    _RailLengthXpu                := _fbXpuPart.GetLength();
    _RailLengthGroup              := _fbMc2CaGroup.GetRailLength();
    _nLengthXpu                   := TO_UINT(_RailLengthXpu);
    _nLengthGroup                 := TO_UINT(_RailLengthGroup);
END_CASE
//-----------------------------------------------------------------------------
//-----------------------------------------------------------------------------
CASE _eState
OF
  //---------------------------------------------------------------------------
  E_PROGRESS.PROGRESS_STARTUP:    // check data for errors
    IF NOT (_bAllPositionsValid)
    THEN
      _eChk                       := E_XPU_CHECK.PROCESSING_UNIT_POSITIONS_VALID;
      _eState := _eResult         := E_PROGRESS.PROGRESS_ERROR;

      _stMsg.eType                := E_MessageType.eMessageError;
      _stMsg.eSubdevice           := e_Subdevice.Xpu_fbProcessingUnit;
      _stMsg.iErrorNumber         := 0;
      _stMsg.sText                := concat(TO_STRING(E_XPU_CHECK.PROCESSING_UNIT_POSITIONS_VALID), ': ');
      _stMsg.sText                := concat(_stMsg.sText, TO_STRING(_eResult));
      f_MessageSet(_stMsg);

    ELSIF NOT (_nLengthXpu > 0)
    THEN
      _eChk                       := E_XPU_CHECK.XPU_RAIL_LENGTH;
      _eState := _eResult         := E_PROGRESS.PROGRESS_ERROR;

      _stMsg.eType                := E_MessageType.eMessageError;
      _stMsg.eSubdevice           := e_Subdevice.Xpu_fbProcessingUnit;
      _stMsg.iErrorNumber         := 0;
      _stMsg.sText                := concat(TO_STRING(E_XPU_CHECK.XPU_RAIL_LENGTH), ': ');
      _stMsg.sText                := concat(_stMsg.sText, TO_STRING(_eResult));
      f_MessageSet(_stMsg);

    ELSIF NOT (_nLengthGroup > 0)
    THEN
      _eChk                       := E_XPU_CHECK.GROUP_RAIL_LENGTH;
      _eState := _eResult         := E_PROGRESS.PROGRESS_ERROR;
     
      _stMsg.eType                := E_MessageType.eMessageError;
      _stMsg.eSubdevice           := e_Subdevice.Xpu_fbProcessingUnit;
      _stMsg.iErrorNumber         := 0;
      _stMsg.sText                := concat(TO_STRING(E_XPU_CHECK.GROUP_RAIL_LENGTH), ': ');
      _stMsg.sText                := concat(_stMsg.sText, TO_STRING(_eResult));
      f_MessageSet(_stMsg);

    ELSIF NOT (_nDetectedMoverCount = _nExpectedMoverCount)
    THEN
      _bMoverIdDetectionValid     := FALSE;
      _eChk                       := E_XPU_CHECK.MOVER_COUNT_NOT_EQUAL;
      _eState := _eResult         := E_PROGRESS.PROGRESS_ERROR;

      _stMsg.eType                := E_MessageType.eMessageError;
      _stMsg.eSubdevice           := e_Subdevice.Xpu_fbProcessingUnit;
      _stMsg.iErrorNumber         := 0;
      _stMsg.sText                := concat(TO_STRING(E_XPU_CHECK.MOVER_COUNT_NOT_EQUAL), ': ');
      _stMsg.sText                := concat(_stMsg.sText, TO_STRING(_eResult));
      f_MessageSet(_stMsg);
  
    ELSIF NOT (_nLengthXpu = _nLengthGroup)
    THEN
      _eChk                       := E_XPU_CHECK.RAIL_LENGTH_COMPARE;
      _eState := _eResult         := E_PROGRESS.PROGRESS_ERROR;
 
      _stMsg.eType                := E_MessageType.eMessageError;
      _stMsg.eSubdevice           := e_Subdevice.Xpu_fbProcessingUnit;
      _stMsg.iErrorNumber         := 0;
      _stMsg.sText                := concat(TO_STRING(E_XPU_CHECK.RAIL_LENGTH_COMPARE), ': ');
      _stMsg.sText                := concat(_stMsg.sText, TO_STRING(_eResult));
      f_MessageSet(_stMsg);

    ELSE
      _eResult                    := E_PROGRESS.PROGRESS_WORKING;

      IF NOT (__ISVALIDREF(_ModuleInfoData))
      THEN
        _eState                   := E_PROGRESS.PROGRESS_BUSY;

        _stMsg.eType              := E_MessageType.eMessageError;
        _stMsg.eSubdevice         := e_Subdevice.Xpu_fbPartModules;
        _stMsg.iErrorNumber       := 0;
        _stMsg.sText              := concat(TO_STRING(_eState), ': ');
        _stMsg.sText              := concat(_stMsg.sText, 'NOT VALID _ModuleInfoData ref');
      ELSE
        _eJobResult               := ModuleInfoData(TRUE);
  
        IF (_eJobResult = E_PROGRESS.PROGRESS_DONE)
        THEN
          _eState                 := E_PROGRESS.PROGRESS_BUSY;
        END_IF  
      END_IF
    END_IF
END_CASE

Cycle                             := _eResult;
END_METHOD

METHOD GetEnvironment : I_TcIoXtsEnvironment
VAR_INPUT
END_VAR
IF NOT (_eInit = E_XPU_INIT.INIT_DONE) THEN RETURN; END_IF

GetEnvironment := _fbEnvironment;
END_METHOD

METHOD GetNctBaseUnit : Tc3_XTS_Utility.I_TcIoXtsNctBaseUnitInterface
VAR_INPUT
  Index     : UINT;
END_VAR
IF NOT (_eInit = E_XPU_INIT.INIT_DONE) THEN RETURN; END_IF

IF NOT (Index > 0) OR
   NOT (Index < MAX_NCT_BASE_UNIT+1)
THEN
  RETURN;
ELSE
  GetNctBaseUnit    := _ItfNctBaseUnit[Index];
END_IF
END_METHOD

METHOD GetNctController : Tc3_XTS_Utility.I_TcIoXtsNctController
VAR_INPUT
END_VAR
IF NOT (_eInit = E_XPU_INIT.INIT_DONE) THEN RETURN; END_IF

GetNctController := _fbNctController;
END_METHOD

METHOD GetParameterSet : I_TcIoXtsParameterSet
VAR_INPUT
  Index     : UINT;
END_VAR
IF NOT (_eInit = E_XPU_INIT.INIT_DONE) THEN RETURN; END_IF

IF NOT (Index > 0) OR
   NOT (Index < MAX_PARAMETER_SET+1)
THEN
  RETURN;
ELSE
  GetParameterSet   := _fbParameterSet[Index];
END_IF
END_METHOD

METHOD GetProcessingUnit : Tc3_XTS_Utility.I_TcIoXtsProcessingUnit
VAR_INPUT
END_VAR
IF NOT (_eInit = E_XPU_INIT.INIT_DONE) THEN RETURN; END_IF

GetProcessingUnit := _fbProcessingUnit;
END_METHOD

METHOD GetXpuMover : Tc3_XTS_Utility.I_TcIoXtsXpuMover
VAR_INPUT
  Index     : UINT;
END_VAR
IF NOT (_eInit = E_XPU_INIT.INIT_DONE) THEN RETURN; END_IF

IF NOT (Index > 0) OR
   NOT (Index < MAX_MOVER+1)
THEN
  RETURN;
ELSE
  GetXpuMover   := _fbMoverXpu[Index];
END_IF
END_METHOD

// mothers' little helper for display in visu
METHOD IdDetectionModeToString : string(20)
VAR
  _DetectionMode    : MoverIdDetectionMode; // Mover ID detection procedure
END_VAR
// just a little helper for visu display
IF NOT (_eInit = E_XPU_INIT.INIT_DONE) THEN IdDetectionModeToString := 'INIT required'; RETURN; END_IF

_DetectionMode := _fbProcessingUnit.GetMoverIdDetectionMode();

CASE _DetectionMode
OF
  MoverIdDetectionMode.Standard:
    IdDetectionModeToString       := 'Standard';

  MoverIdDetectionMode.Mover1:
    IdDetectionModeToString       := 'Mover 1';

  MoverIdDetectionMode.MultipleMover1:
    IdDetectionModeToString       := 'Multiple Mover 1';

ELSE
    IdDetectionModeToString       := 'UNKNOWN Mode';
END_CASE
END_METHOD

PROPERTY MessageLevel : e_messagetype
SET
_eMessageLevel := MessageLevel;
END_SET
END_PROPERTY

// mothers' little helper for display in visu
METHOD PRIVATE ModuleInfoData : E_PROGRESS
VAR_INPUT
  Enable        : BOOL; // enable to read ST_InfoDataView for diag/display
END_VAR
VAR_INST
  _idt,
  _nModule : UINT;
  _eReturn,
  _eState       : E_PROGRESS;
  _aPcbTemp     : ARRAY[1..4] OF REAL;
END_VAR
//---------------------------------------------------------------------------------------------
// just a little helper for visu display
// collects module data for local data
//---------------------------------------------------------------------------------------------
IF NOT (_eInit = E_XPU_INIT.INIT_DONE)      // if Xpu init is not done, just leave
THEN 
  RETURN; 
END_IF
//---------------------------------------------------------------------------------------------
IF NOT Enable                               // clear states on request
THEN
  _eReturn                                  := 
  _eState                                   := E_PROGRESS.PROGRESS_INIT; 
END_IF 
//---------------------------------------------------------------------------------------------
IF NOT (__ISVALIDREF(_ModuleInfoData))      // datafield not connected, error and leave
THEN
  ModuleInfoData                            := E_PROGRESS.PROGRESS_ERROR;
  RETURN;
END_IF
//---------------------------------------------------------------------------------------------
CASE _eState                                // get InfoData from motor modules
OF
  //-------------------------------------------------------------------------------------------
  E_PROGRESS.PROGRESS_INIT:
    IF Enable
    THEN
      _eState                                             := E_PROGRESS.PROGRESS_BUSY;
      _nModule                                            := 1;
    END_IF
END_CASE
CASE _eState
OF
  //-------------------------------------------------------------------------------------------
  E_PROGRESS.PROGRESS_BUSY:
    _eState                                               := E_PROGRESS.PROGRESS_PREPARE;

    _ModuleInfoData[_nModule].fAuxiliaryVoltage_5V        := _fbPartModules[_nModule].GetAuxiliaryVoltage5V();
    _ModuleInfoData[_nModule].fAuxiliaryVoltage_10V       := _fbPartModules[_nModule].GetAuxiliaryVoltage10V();
    _ModuleInfoData[_nModule].fAuxiliaryVoltage_24V       := _fbPartModules[_nModule].GetAuxiliaryVoltage24V();

    _ModuleInfoData[_nModule].fDcLinkVoltage              := _fbPartModules[_nModule].GetDCLinkVoltage();

    IF (_ModuleInfoData[_nModule].fDcLinkVoltage > 48.0*0.85) AND
       (_ModuleInfoData[_nModule].fDcLinkVoltage < 48.0*1.15)
    THEN
      _bModulePower[_nModule]                             := TRUE;
    ELSE
      _bModulePower[_nModule]                             := SEL((_XpuOperationMode = OperationMode.Simulation), FALSE, TRUE);
    END_IF

    _ModuleInfoData[_nModule].nCurrentScaling             := TO_INT(_fbPartModules[_nModule].GetCurrentScaling());

    _ModuleInfoData[_nModule].nDeviceInfo                 := _fbPartModules[_nModule].GetDeviceInfo();

    IF (_XpuOperationMode = OperationMode.Normal)
    THEN
      _ModuleInfoData[_nModule].fAverageTemp              := 0.0;
  
      _aPcbTemp                                           := _fbPartModules[_nModule].GetPCBTemperatures();
  
      _ModuleInfoData[_nModule].fPcbTemp_0                := _aPcbTemp[1];
      _ModuleInfoData[_nModule].fPcbTemp_1                := _aPcbTemp[2];
      _ModuleInfoData[_nModule].fPcbTemp_2                := _aPcbTemp[3];
      _ModuleInfoData[_nModule].fPcbTemp_3                := _aPcbTemp[4];

      FOR _idt := 1 TO 4
      DO
        _ModuleInfoData[_nModule].fAverageTemp            := _ModuleInfoData[_nModule].fAverageTemp + _aPcbTemp[_idt];
      END_FOR
      _ModuleInfoData[_nModule].fAverageTemp              := _ModuleInfoData[_nModule].fAverageTemp / 4;
    END_IF

    _ModuleInfoData[_nModule].fOverallCurrent             := _fbPartModules[_nModule].GetOverallCurrent();

    _ModuleInfoData[_nModule].fMaxDCLinkVoltageLast500ms  := _fbPartModules[_nModule].GetMaxDCLinkVoltageLast500ms();
    _ModuleInfoData[_nModule].fMaxOverallCurrentLast500ms := _fbPartModules[_nModule].GetMaxOverallCurrentLast500ms();
END_CASE
CASE _eState 
OF
  //-------------------------------------------------------------------------------------------
  E_PROGRESS.PROGRESS_PREPARE:
    IF (_nModule > _nModuleCount-1)
    THEN
      _eState                                             := E_PROGRESS.PROGRESS_WORKING;
    ELSE
      _nModule                                            := _nModule + 1;
      _eReturn                                            :=
      _eState                                             := E_PROGRESS.PROGRESS_BUSY;
    END_IF

  //-------------------------------------------------------------------------------------------
  E_PROGRESS.PROGRESS_WORKING:
    _eReturn                                              := E_PROGRESS.PROGRESS_DONE;
    _eState                                               := E_PROGRESS.PROGRESS_INIT;
END_CASE

ModuleInfoData                                            := _eReturn;
END_METHOD

// mothers' little helper for display in visu
METHOD MoverPositionAssignementToString : string(20)
VAR
  _PositionAssignement    : MoverPositionAssignment; // XPU movver assignement procedure
END_VAR
// just a little helper for visu display
IF NOT (_eInit = E_XPU_INIT.INIT_DONE) THEN MoverPositionAssignementToString := 'INIT required'; RETURN; END_IF

_PositionAssignement      := _fbProcessingUnit.GetMoverPositionAssignment();

CASE _PositionAssignement
OF
  MoverPositionAssignment.Standard:
    MoverPositionAssignementToString    := 'Standard';

  MoverPositionAssignment.StartAtFirstMover:
    MoverPositionAssignementToString    := 'Start At First Mover';
ELSE
    MoverPositionAssignementToString    := 'UNKNOWN Assgnement';
END_CASE
END_METHOD

// mothers' little helper for display in visu
METHOD OpModeToString : String(20)
VAR
  _OpMode     : OperationMode; // XPU operation mode
END_VAR
// just a little helper for visu display
IF NOT (_eInit = E_XPU_INIT.INIT_DONE) THEN OpModeToString := 'INIT required'; RETURN; END_IF

_OpMode   := _fbProcessingUnit.GetOperationMode();

CASE _OpMode
OF
  OperationMode.Normal:
    OpModeToString      := 'Normal';

  OperationMode.Simulation:
    OpModeToString      := 'Simulation';

ELSE
    OpModeToString      := 'UNKNOWN OP MODE';
END_CASE
END_METHOD

PROPERTY RailLength : lreal
GET
IF (_eInit = E_XPU_INIT.INIT_DONE)
THEN
  RailLength := _fbXpuPart.GetLength();
ELSE
  RailLength := 0.0;
END_IF
END_GET
END_PROPERTY

PROPERTY XpuInfo : st_xpu_info
GET
IF NOT (_eInit = E_XPU_INIT.INIT_DONE) THEN RETURN; END_IF

_XpuInfo.AllPositionsValid        := _bAllPositionsValid;

_XpuInfo.IdDetectionError         := _bMoverIdDetectionError;
_XpuInfo.IdDetectionValid         := _bMoverIdDetectionValid;

_XpuInfo.IdDetectionActive        := _fbProcessingUnit.GetIsMoverIdDetectionActive();

_XpuInfo.OperationMode            := TO_UINT(_fbProcessingUnit.GetOperationMode());

_XpuInfo.IdDetectionMode          := TO_UINT(_fbProcessingUnit.GetMoverIdDetectionMode());
_XpuInfo.MoverPositionAssignement := TO_UINT(_fbProcessingUnit.GetMoverPositionAssignment());

_XpuInfo.nDetectedAxisCount       := _nDetectedMoverCount;
_XpuInfo.nExpectedAxisCount       := _nExpectedMoverCount;

_XpuInfo.nParameterSetCount       := _nParameterSetCount;

XpuInfo := _XpuInfo;
END_GET
END_PROPERTY

METHOD PROTECTED XpuInit  : E_XPU_INIT      // connect to TcCOM
VAR_INPUT
  Execute       : BOOL;           // must be executed for connecting to TcCOM Environment of Xpu
END_VAR
VAR_IN_OUT
  _eReslt       : E_PROGRESS;     // send info about progress to caller
  _eChk         : E_XPU_CHECK;
END_VAR
VAR_INST
  _eState           : E_PROGRESS;   // progress state
  _nState           : E_XPU_INIT;   // initialization state
  _eDataGetCount    : E_PROGRESS;   // cycle counter to catch exceeding wait time for data from ProcessingUnit

  _nParaSetIdx      : UINT;

  _nMoverIdx,
  _nModuleIdx       : UINT;

  _nNctBaseUnitIdx        : UINT;
END_VAR
//-----------------------------------------------------------------------------------------------
//-----------------------------------------------------------------------------------------------
// clear progress on request
IF NOT Execute 
THEN 
  _eState                           := E_PROGRESS.PROGRESS_INIT;
  _eDataGetCount                    := 0;
 
  XpuInit                           :=
  _nState                           := E_XPU_INIT.INIT_START; 
  RETURN; 
END_IF
//-----------------------------------------------------------------------------------------------
//-----------------------------------------------------------------------------------------------
// progress state
//-----------------------------------------------------------------------------------------------
//-----------------------------------------------------------------------------------------------
CASE _eState
OF
  E_PROGRESS.PROGRESS_INIT:         // clear start
    IF Execute
    THEN
      _eState                       := E_PROGRESS.PROGRESS_BUSY;
      _eChk                         := E_XPU_CHECK.INIT_CHECK;    // clear cyclic check state
      _sVersionNctController        :=
      _sVersionXpu                  := TO_STRING(_eChk);          // clear Version string

      // always initialize environment function blocks to get defined start of progress
      _fbEnvironment.Init(FALSE);
      _fbEnvironment.GetXpuOids(FALSE);
      _fbEnvironment.GetInfoServerOids(FALSE);

      // clear initialization states
      _nState                       := E_XPU_INIT.INIT_START;

      // clear check bits
      _bAllPositionsValid           :=
      _bMoverIdDetectionValid       :=
      _bMoverIdDetectionError       := FALSE;

      // clear check values
      _nLengthXpu                   :=
      _nLengthGroup                 :=
      _nDetectedMoverCount          :=
      _nExpectedMoverCount          := 0;

      // clear work values
      _nNctBaseUnitCount            :=
      _nNctBaseUnitIdx              :=
      _nParameterSetCount           :=
      _nInfoServerCount             :=
      _nIfoStationCount             :=
      _nPartCount                   :=
      _nTrackCount                  :=
      _nTaskCount                   :=
      _nMoverCount                  :=
      _nModuleCount                 :=
      _nMoverIdx                    :=
      _nModuleIdx                   := 0;

      IF (_eMessageLevel = E_MessageType.eMessageVerbose)
      THEN
        _stMsg.eType                := E_MessageType.eMessageVerbose;
        _stMsg.eSubdevice           := e_Subdevice.Xpu_fbEnvironment;
        _stMsg.iErrorNumber         := 0;
        _stMsg.sText                := concat(TO_STRING(_eState), ': ');
        _stMsg.sText                := concat(_stMsg.sText, TO_STRING(_eChk));
        f_MessageSet(_stMsg);
      END_IF
    END_IF
END_CASE
//-----------------------------------------------------------------------------------------------
//-----------------------------------------------------------------------------------------------
//-----------------------------------------------------------------------------------------------
CASE _eState
OF
  E_PROGRESS.PROGRESS_BUSY:         // begin with initializing environment
    CASE _nState
    OF
  //-----------------------------------------------------------------------------------------------
  //-----------------------------------------------------------------------------------------------
  INIT_START:                       // call initialization of environment

    IF NOT _fbEnvironment.P_IsInitialized
    THEN
      _fbEnvironment.Init(TRUE);
    END_IF

    IF (_fbEnvironment.bError)
    THEN
      _eChk                         := E_XPU_CHECK.INIT_CHECK_ERROR;
                                    
      _stMsg.eType                  := E_MessageType.eMessageError;
      _stMsg.eSubdevice             := e_Subdevice.Xpu_fbEnvironment;
      _stMsg.iErrorNumber           := 666;
      _stMsg.sText                  := concat(TO_STRING(_eState), ': ');
      _stMsg.sText                  := concat(_stMsg.sText, TO_STRING(_eChk));
      f_MessageSet(_stMsg);

      _eState                       := E_PROGRESS.PROGRESS_ERROR;

    // get information about success in Property (P_<function>)
    ELSIF _fbEnvironment.P_IsInitialized
    THEN
      // now environment is initialized
     
      //---------------------------------------------------------------------
      // use of local function block instances
      // get information about Object IDs to local datafields
      //---------------------------------------------------------------------
      //  - everything else in this state machine is for use within fb_Xpu
      //  - the following states shall illustrate how TcCOM Objects are connected through XTS_Utility lib
      //  - local instances of members of Environment are connected from here onward
      //
      IF _fbEnvironment.GetXpuOids(TRUE) // get object IDs for all processing units
      THEN
        _fbEnvironment.Init(FALSE);// clear environment init
        _nState                     := INIT_ENVIRONMENT_OID;

        IF (_eMessageLevel = E_MessageType.eMessageVerbose)
        THEN
          _stMsg.eType              := E_MessageType.eMessageVerbose;
          _stMsg.eSubdevice         := e_Subdevice.Xpu_fbEnvironment;
          _stMsg.iErrorNumber       := 0;
          _stMsg.sText              := concat(TO_STRING(_eState), ': ');
          _stMsg.sText              := concat(_stMsg.sText, TO_STRING(_nState));
          f_MessageSet(_stMsg);
        END_IF
      END_IF
    END_IF

  //-----------------------------------------------------------------------------------------------
  //-----------------------------------------------------------------------------------------------
  INIT_ENVIRONMENT_OID:             // get processing unit object ID for THIS instance
    _Xpu_OTCID                      := _fbEnvironment.P_XpuOids[_nXpu];   // fb_Xpu.XpuInstance --> _nXpu

    // clear all local object IDs
    memset(ADR(_Part_OTCID)         , 0, SIZEOF(_Part_OTCID));
    memset(ADR(_Track_OTCID)        , 0, SIZEOF(_Track_OTCID));
    memset(ADR(_Mov_OTCID)          , 0, SIZEOF(_Mov_OTCID));
    memset(ADR(_Module_OTCID)       , 0, SIZEOF(_Module_OTCID));
    memset(ADR(_ParameterSet_OTCID) , 0, SIZEOF(_ParameterSet_OTCID));

    // clear function blocks
    _fbEnvironment.GetXpuOids           (FALSE);
    _fbEnvironment.GetCaGroupCount      (FALSE);
    _fbEnvironment.GetInfoServerCount   (FALSE);
    _fbEnvironment.GetParameterSetCount (FALSE);

    _eState                         := E_PROGRESS.PROGRESS_PREPARE; // TODO - implement InfoServer R/W
    _nState                         := INIT_CA_GROUP_OID;           // TODO - implement initialization states for info server procedure

    //_nState                       := INIT_INFO_SERVER_ITF;              // check environment for info servers

  //-----------------------------------------------------------------------------------------------
  //-----------------------------------------------------------------------------------------------
  INIT_INFO_SERVER_ITF:           // HAUD 2024 03 14: TODO - implement procedure for getting Info server data to local datafields
    IF _fbEnvironment.GetInfoServerCount(TRUE)
    THEN
      // how many of you are there?
      _nInfoServerCount             := _fbEnvironment.P_InfoServerCount;

      IF (_nInfoServerCount > 0)
      THEN
        // go do something with the data
        //
        //  TODO - get station coordinates
        _eState                     := E_PROGRESS.PROGRESS_PREPARE; // TODO - implement InfoServer R/W
        _nState                     := INIT_CA_GROUP_OID;           // TODO - implement initialization states for info server procedure

        IF (_eMessageLevel = E_MessageType.eMessageVerbose)
        THEN
          _stMsg.eType              := E_MessageType.eMessageVerbose;
          _stMsg.eSubdevice         := e_Subdevice.Xpu_fbEnvironment;
          _stMsg.iErrorNumber       := 0;
          _stMsg.sText              := concat(TO_STRING(_eState), ': ');
          _stMsg.sText              := concat(_stMsg.sText, TO_STRING(_nState));
          f_MessageSet(_stMsg);
        END_IF

      ELSE
        // no info server present
        _eState                     := E_PROGRESS.PROGRESS_PREPARE;
        _nState                     := INIT_CA_GROUP_OID; // go check CA group

        IF (_eMessageLevel = E_MessageType.eMessageVerbose)
        THEN
          _stMsg.eType              := E_MessageType.eMessageVerbose;
          _stMsg.eSubdevice         := e_Subdevice.Xpu_fbEnvironment;
          _stMsg.iErrorNumber       := 0;
          _stMsg.sText              := concat(TO_STRING(_eState), ': ');
          _stMsg.sText              := concat(_stMsg.sText, TO_STRING(_nState));
          f_MessageSet(_stMsg);
        END_IF
      END_IF
    END_IF
  END_CASE
END_CASE
//-----------------------------------------------------------------------------------------------
//-----------------------------------------------------------------------------------------------
//-----------------------------------------------------------------------------------------------
CASE _eState
OF
  E_PROGRESS.PROGRESS_PREPARE:      // CA group initialization
  CASE _nState
  OF
  //-----------------------------------------------------------------------------------------------
  //-----------------------------------------------------------------------------------------------
  INIT_CA_GROUP_OID:                // get object IDs of all CA groups in environment
    IF _fbEnvironment.GetCaGroupOids(TRUE)
    THEN
      _Group_OTCID                  := _fbEnvironment.P_CaGroupOids;  // copy all Ids to local
      _nState                       := INIT_CA_GROUP_GET_OID;

      IF (_eMessageLevel = E_MessageType.eMessageVerbose)
      THEN
        _stMsg.eType                := E_MessageType.eMessageVerbose;
        _stMsg.eSubdevice           := e_Subdevice.Xpu_fbEnvironment;
        _stMsg.iErrorNumber         := 0;
        _stMsg.sText                := concat(TO_STRING(_eState), ': ');
        _stMsg.sText                := concat(_stMsg.sText, TO_STRING(_nState));
        f_MessageSet(_stMsg);
      END_IF
    END_IF

  //-----------------------------------------------------------------------------------------------
  //-----------------------------------------------------------------------------------------------
  INIT_CA_GROUP_GET_OID:            // look for any CA group
    _fbEnvironment.GetCaGroupOids(FALSE);
    IF NOT (_Group_OTCID[1] <> 0)
    THEN
      // no group is configured in project --> error, go add/link CA Group in NC objects
      _eChk                         := E_XPU_CHECK.GROUP_NOT_CONFIGURED;
      _eState                       := E_PROGRESS.PROGRESS_ERROR;

      _stMsg.eType                  := E_MessageType.eMessageError;
      _stMsg.eSubdevice             := e_Subdevice.Xpu_fbEnvironment;
      _stMsg.iErrorNumber           := 0;
      _stMsg.sText                  := concat(TO_STRING(_eState), ': ');
      _stMsg.sText                  := concat(_stMsg.sText, TO_STRING(_nState));
      f_MessageSet(_stMsg);
    ELSE
      _nState                       := INIT_CA_GROUP_CHECK_OID; // get matching CA group

      IF (_eMessageLevel = E_MessageType.eMessageVerbose)
      THEN
        _stMsg.eType                := E_MessageType.eMessageVerbose;
        _stMsg.eSubdevice           := e_Subdevice.Xpu_fbEnvironment;
        _stMsg.iErrorNumber         := 0;
        _stMsg.sText                := concat(TO_STRING(_eState), ': ');
        _stMsg.sText                := concat(_stMsg.sText, TO_STRING(_nState));
        //f_MessageSet(_stMsg);
      END_IF
    END_IF

  //-----------------------------------------------------------------------------------------------
  //-----------------------------------------------------------------------------------------------
  INIT_CA_GROUP_CHECK_OID:          // ID must be found, there is one chance
    _eChk                           := E_XPU_CHECK.GROUP_OID_MISMATCH;
    _eState                         := E_PROGRESS.PROGRESS_ERROR;

    FOR _ix := 1 TO MAX_GROUP
    DO
      IF (_fbEnvironment.P_CaGroupOids[_ix] <> 0)
      THEN
        // check whether the input from cyclic interface can be found in XPU data
        IF (_fbEnvironment.P_CaGroupOids[_ix] = _CaGroupOID)  // _CaGroupOID must be linked from NC Objects into PLC (GROUP_REF)
        THEN

          _eState                   := E_PROGRESS.PROGRESS_PREPARE; // stay here
          _eChk                     := E_XPU_CHECK.INIT_CHECK;

          _nGroup                   := _ix;

          _fbEnvironment.GetCaGroupOids(FALSE);
          _nState                   := INIT_CA_GROUP_COM; // only continue if match was found

          IF (_eMessageLevel = E_MessageType.eMessageVerbose)
          THEN
            _stMsg.eType            := E_MessageType.eMessageVerbose;
            _stMsg.eSubdevice       := e_Subdevice.Xpu_fbEnvironment;
            _stMsg.iErrorNumber     := _CaGroupOID;
            _stMsg.sText            := concat(TO_STRING(_eState), ': ');
            _stMsg.sText            := concat(_stMsg.sText, TO_STRING(_nState));
            f_MessageSet(_stMsg);
          END_IF
          EXIT;
        END_IF
      END_IF
    END_FOR

    IF (_eState = E_PROGRESS.PROGRESS_ERROR)
    THEN
      _stMsg.eType                  := E_MessageType.eMessageError;
      _stMsg.eSubdevice             := e_Subdevice.Xpu_fbEnvironment;
      _stMsg.iErrorNumber           := _nGroup;
      _stMsg.sText                  := concat(TO_STRING(_eState), ': ');
      _stMsg.sText                  := concat(_stMsg.sText, TO_STRING(_nState));
      f_MessageSet(_stMsg);
    END_IF

  //-----------------------------------------------------------------------------------------------
  //-----------------------------------------------------------------------------------------------
  INIT_CA_GROUP_COM:                // connect to CaGroup function block in environment
    IF (_fbMc2CaGroup.GetComObject(_fbEnvironment.P_CaGroupOids[_nGroup]))
    THEN
      _fbEnvironment.GetParameterSetCount(FALSE);

      _nState                       := INIT_PARAMETERSET_COUNT;

      IF (_eMessageLevel = E_MessageType.eMessageVerbose)
      THEN
        _stMsg.eType                := E_MessageType.eMessageVerbose;
        _stMsg.eSubdevice           := e_Subdevice.Xpu_fbEnvironment;
        _stMsg.iErrorNumber         := _nGroup;
        _stMsg.sText                := concat(TO_STRING(_eState), ': ');
        _stMsg.sText                := concat(_stMsg.sText, TO_STRING(_nState));
       f_MessageSet(_stMsg);
      END_IF
    END_IF

  //-----------------------------------------------------------------------------------------------
  //-----------------------------------------------------------------------------------------------
  INIT_PARAMETERSET_COUNT:
    IF _fbEnvironment.GetParameterSetCount(TRUE)
    THEN
      _fbEnvironment.GetParameterSetOids(FALSE);
      _nParaSetIdx                  :=
      _nParameterSetCount           := _fbEnvironment.P_ParameterSetCount;
      _nState                       := INIT_PARAMETERSET_OID; 

      IF (_eMessageLevel = E_MessageType.eMessageVerbose)
      THEN
        _stMsg.eType                := E_MessageType.eMessageVerbose;
        _stMsg.eSubdevice           := e_Subdevice.Xpu_fbEnvironment;
        _stMsg.iErrorNumber         := _nParameterSetCount;
        _stMsg.sText                := concat(TO_STRING(_eState), ': ');
        _stMsg.sText                := concat(_stMsg.sText, TO_STRING(_nState));
        f_MessageSet(_stMsg);
      END_IF
    END_IF

  //-----------------------------------------------------------------------------------------------
  //-----------------------------------------------------------------------------------------------
  INIT_PARAMETERSET_OID:
    IF (_nParameterSetCount = 0)
    THEN
      _fbEnvironment.GetParameterSetCount(FALSE);
      _eState                       := E_PROGRESS.PROGRESS_STARTUP;
      _nState                       := INIT_PROCESSING_UNIT_COM;

    ELSIF _fbEnvironment.GetParameterSetOids(TRUE)
    THEN
      _fbEnvironment.GetParameterSetCount(FALSE);
      _ParameterSet_OTCID           := _fbEnvironment.P_ParameterSetOids;
      _nState                       := INIT_PARAMETERSET_COM;
    END_IF

  //-----------------------------------------------------------------------------------------------
  //-----------------------------------------------------------------------------------------------
  INIT_PARAMETERSET_COM:
    IF (_nParaSetIdx > 0)
    THEN
      IF _fbParameterSet[_nParaSetIdx].GetComObject(_ParameterSet_OTCID[_nParaSetIdx])
      THEN
        _nState                     := INIT_PARAMETERSET_COM_NEXT;

        IF (_eMessageLevel = E_MessageType.eMessageVerbose)
        THEN
          _stMsg.eType              := E_MessageType.eMessageVerbose;
          _stMsg.eSubdevice         := e_Subdevice.Xpu_fbParameterSet;
          _stMsg.iErrorNumber       := _ParameterSet_OTCID[_nParaSetIdx];
          _stMsg.sText              := concat(TO_STRING(_eState), ': ');
          _stMsg.sText              := concat(_stMsg.sText, TO_STRING(_nState));
          f_MessageSet(_stMsg);
        END_IF
      END_IF
    ELSE
      _fbEnvironment.GetParameterSetOids(FALSE);
      _eState                       := E_PROGRESS.PROGRESS_STARTUP;
      _nState                       := INIT_PROCESSING_UNIT_COM;
    END_IF
      

  //-----------------------------------------------------------------------------------------------
  //-----------------------------------------------------------------------------------------------
  INIT_PARAMETERSET_COM_NEXT:
    _nParaSetIdx                    := _nParaSetIdx - 1;
    _nState                         := INIT_PARAMETERSET_COM; 
  END_CASE
END_CASE
//-----------------------------------------------------------------------------------------------
//-----------------------------------------------------------------------------------------------
//-----------------------------------------------------------------------------------------------
CASE _eState
OF
  E_PROGRESS.PROGRESS_STARTUP:      // ProcessingUnit initialization
  CASE _nState
  OF
  //-----------------------------------------------------------------------------------------------
  //-----------------------------------------------------------------------------------------------
  INIT_PROCESSING_UNIT_COM:         // connect local function block with TcCom object
    IF (_fbProcessingUnit.GetComObject(_Xpu_OTCID))
    THEN
      // local function block can now be used to get information
      // get operation mode first
      _XpuOperationMode             := _fbProcessingUnit.GetOperationMode();
      _nState                       := INIT_PROCESSING_UNIT_PART_COUNT;

      IF (_eMessageLevel = E_MessageType.eMessageVerbose)
      THEN
        _stMsg.eType                := E_MessageType.eMessageVerbose;
        _stMsg.eSubdevice           := e_Subdevice.Xpu_fbProcessingUnit;
        _stMsg.iErrorNumber         := _nGroup;
        _stMsg.sText                := concat(TO_STRING(_eState), ': ');
        _stMsg.sText                := concat(_stMsg.sText, TO_STRING(_nState));
        f_MessageSet(_stMsg);
      END_IF
    END_IF

  //-----------------------------------------------------------------------------------------------
  //-----------------------------------------------------------------------------------------------
  INIT_PROCESSING_UNIT_PART_COUNT:  // get parts in ProcessingUnit
    _nPartCount                     := TO_UINT(_fbProcessingUnit.GetPartCount());

    IF (_nPartCount > 0)            // one is enough
    THEN
      _nState                       := INIT_PROCESSING_UNIT_PART_OID;

      IF (_eMessageLevel = E_MessageType.eMessageVerbose)
      THEN
        _stMsg.eType                := E_MessageType.eMessageVerbose;
        _stMsg.eSubdevice           := e_Subdevice.Xpu_fbProcessingUnit;
        _stMsg.iErrorNumber         := _nGroup;
        _stMsg.sText                := concat(TO_STRING(_eState), ': ');
        _stMsg.sText                := concat(_stMsg.sText, TO_STRING(_nState));
        f_MessageSet(_stMsg);
      END_IF
    END_IF

  //-----------------------------------------------------------------------------------------------
  //-----------------------------------------------------------------------------------------------
  INIT_PROCESSING_UNIT_PART_OID:    // get object IDs of all parts in ProcessingUNit
    IF _fbProcessingUnit.GetPartOids()
    THEN
      _Part_OTCID                   := _fbProcessingUnit.P_PartOids;  // copy IDs to local
      _nState                       := INIT_PROCESSING_UNIT_TRACK_COUNT;

      IF (_eMessageLevel = E_MessageType.eMessageVerbose)
      THEN
        _stMsg.eType                := E_MessageType.eMessageVerbose;
        _stMsg.eSubdevice           := e_Subdevice.Xpu_fbProcessingUnit;
        _stMsg.iErrorNumber         := _nGroup;
        _stMsg.sText                := concat(TO_STRING(_eState), ': ');
        _stMsg.sText                := concat(_stMsg.sText, TO_STRING(_nState));
        f_MessageSet(_stMsg);
      END_IF
    END_IF

  //-----------------------------------------------------------------------------------------------
  //-----------------------------------------------------------------------------------------------
  INIT_PROCESSING_UNIT_TRACK_COUNT: // how many tracks does this ProcessingUnit have?
    _nTrackCount                    := TO_UINT(_fbProcessingUnit.GetTrackCount());
  
    IF (_nTrackCount > 0)           // one is enough
    THEN
      _nState                       := INIT_PROCESSING_UNIT_TRACK_OID;

      IF (_eMessageLevel = E_MessageType.eMessageVerbose)
      THEN
        _stMsg.eType                := E_MessageType.eMessageVerbose;
        _stMsg.eSubdevice           := e_Subdevice.Xpu_fbProcessingUnit;
        _stMsg.iErrorNumber         := _nTrackCount;
        _stMsg.sText                := concat(TO_STRING(_eState), ': ');
        _stMsg.sText                := concat(_stMsg.sText, TO_STRING(_nState));
        f_MessageSet(_stMsg);
      END_IF
    END_IF

  //-----------------------------------------------------------------------------------------------
  //-----------------------------------------------------------------------------------------------
  INIT_PROCESSING_UNIT_TRACK_OID:   // get object IDs of all tracks in ProcessingUnit
    IF _fbProcessingUnit.GetTrackOids()
    THEN
      _Track_OTCID                  := _fbProcessingUnit.P_TrackOids; // copy IDs to local
      _nState                       := INIT_PROCESSING_UNIT_MOVER_COUNT;

      IF (_eMessageLevel = E_MessageType.eMessageVerbose)
      THEN
        _stMsg.eType                := E_MessageType.eMessageVerbose;
        _stMsg.eSubdevice           := e_Subdevice.Xpu_fbProcessingUnit;
        _stMsg.iErrorNumber         := 0;
        _stMsg.sText                := concat(TO_STRING(_eState), ': ');
        _stMsg.sText                := concat(_stMsg.sText, TO_STRING(_nState));
        f_MessageSet(_stMsg);
      END_IF
    END_IF

  //-----------------------------------------------------------------------------------------------
  //-----------------------------------------------------------------------------------------------
  INIT_PROCESSING_UNIT_MOVER_COUNT: // how many of you are there?
    _nMoverCount                    := TO_UINT(_fbProcessingUnit.GetMoverCount());
  
    IF (_nMoverCount > 0)           // one is enough
    THEN
      _nState                       := INIT_PROCESSING_UNIT_MOVER_OID;

      IF (_eMessageLevel = E_MessageType.eMessageVerbose)
      THEN
        _stMsg.eType                := E_MessageType.eMessageVerbose;
        _stMsg.eSubdevice           := e_Subdevice.Xpu_fbProcessingUnit;
        _stMsg.iErrorNumber         := _nMoverCount;
        _stMsg.sText                := concat(TO_STRING(_eState), ': ');
        _stMsg.sText                := concat(_stMsg.sText, TO_STRING(_nState));
        f_MessageSet(_stMsg);
      END_IF
    END_IF

  //-----------------------------------------------------------------------------------------------
  //-----------------------------------------------------------------------------------------------
  INIT_PROCESSING_UNIT_MOVER_OID:   // get object IDs of all mover in ProcessingUnit
    IF _fbProcessingUnit.GetMoverOids()
    THEN
      _Mov_OTCID                    := _fbProcessingUnit.P_MoverOids; // copy IDs to local
      _nState                       := INIT_PROCESSING_UNIT_TASK_COUNT;
      _eChk                         := E_XPU_CHECK.MOVER_COUNT;

      IF (_eMessageLevel = E_MessageType.eMessageVerbose)
      THEN
        _stMsg.eType                := E_MessageType.eMessageVerbose;
        _stMsg.eSubdevice           := e_Subdevice.Xpu_fbProcessingUnit;
        _stMsg.iErrorNumber         := 0;
        _stMsg.sText                := concat(TO_STRING(_eState), ': ');
        _stMsg.sText                := concat(_stMsg.sText, TO_STRING(_nState));
        f_MessageSet(_stMsg);
      END_IF
    END_IF

  //-----------------------------------------------------------------------------------------------
  //-----------------------------------------------------------------------------------------------
  INIT_PROCESSING_UNIT_TASK_COUNT:  // how many?
    _nTaskCount                     := TO_UINT(_fbProcessingUnit.GetTaskCount());
  
    IF (_nTaskCount > 0)
    THEN
      _nState                       := INIT_PROCESSING_UNIT_TASK_OID;

      IF (_eMessageLevel = E_MessageType.eMessageVerbose)
      THEN
        _stMsg.eType                := E_MessageType.eMessageVerbose;
        _stMsg.eSubdevice           := e_Subdevice.Xpu_fbProcessingUnit;
        _stMsg.iErrorNumber         := _nTaskCount;
        _stMsg.sText                := concat(TO_STRING(_eState), ': ');
        _stMsg.sText                := concat(_stMsg.sText, TO_STRING(_nState));
        f_MessageSet(_stMsg);
      END_IF
    END_IF    

  //-----------------------------------------------------------------------------------------------
  //-----------------------------------------------------------------------------------------------
  INIT_PROCESSING_UNIT_TASK_OID:    // get their names!
    IF _fbProcessingUnit.GetTaskOids()
    THEN
      _eState                       := E_PROGRESS.PROGRESS_CHECK;
      _nState                       := INIT_NCT_CONTROLLER_OID;

      IF (_eMessageLevel = E_MessageType.eMessageVerbose)
      THEN
        _stMsg.eType                := E_MessageType.eMessageVerbose;
        _stMsg.eSubdevice           := e_Subdevice.Xpu_fbNctController;
        _stMsg.iErrorNumber         := _nTrack;
        _stMsg.sText                := concat(TO_STRING(_eState), ': ');
        _stMsg.sText                := concat(_stMsg.sText, TO_STRING(_nState));
        f_MessageSet(_stMsg);
      END_IF
    END_IF
  END_CASE
END_CASE
//-----------------------------------------------------------------------------------------------
//-----------------------------------------------------------------------------------------------
//-----------------------------------------------------------------------------------------------
CASE _eState
OF
  E_PROGRESS.PROGRESS_CHECK:        // NCT
  CASE _nState
  OF
  //-----------------------------------------------------------------------------------------------
  //-----------------------------------------------------------------------------------------------
  INIT_NCT_CONTROLLER_OID:
    IF (_fbProcessingUnit.GetNctControllerOid())
    THEN
      _Nct_OTCID                    := _fbProcessingUnit.P_NctControllerOid;

      IF NOT(_Nct_OTCID > 0)
      THEN
        _eState                     := E_PROGRESS.PROGRESS_OCCUPIED;
      ELSE
        _eState                     := E_PROGRESS.PROGRESS_CHECK;
        _nState                     := INIT_NCT_CONTROLLER_COM;

        IF (_eMessageLevel = E_MessageType.eMessageVerbose)
        THEN
          _stMsg.eType              := E_MessageType.eMessageVerbose;
          _stMsg.eSubdevice         := e_Subdevice.Xpu_fbNctController;
          _stMsg.iErrorNumber       := 0;
          _stMsg.sText              := concat(TO_STRING(_eState), ': ');
          _stMsg.sText              := concat(_stMsg.sText, TO_STRING(_nState));
          f_MessageSet(_stMsg);
        END_IF
      END_IF
    END_IF

  //-----------------------------------------------------------------------------------------------
  //-----------------------------------------------------------------------------------------------
  INIT_NCT_CONTROLLER_COM:
    IF (_fbNctController.GetComObject(_Nct_OTCID))
    THEN
      _sVersionNctController        := _fbNctController.GetVersionString();
      _nState                       := INIT_NCT_BASE_UNIT_COUNT;

      IF (_eMessageLevel = E_MessageType.eMessageVerbose)
      THEN
        _stMsg.eType                := E_MessageType.eMessageVerbose;
        _stMsg.eSubdevice           := e_Subdevice.Xpu_fbNctController;
        _stMsg.iErrorNumber         := 0;
        _stMsg.sText                := concat(TO_STRING(_eState), ': ');
        _stMsg.sText                := concat(_stMsg.sText, TO_STRING(_nState));
        f_MessageSet(_stMsg);
      END_IF
      IF (_eMessageLevel > E_MessageType.eMessageError)
      THEN
        _stMsg.eType                := E_MessageType.eMessageInfo;
        _stMsg.eSubdevice           := e_Subdevice.Xpu_fbNctController;
        _stMsg.iErrorNumber         := 0;
        _stMsg.sText                := concat('NctController VersionString: ', _sVersionNctController);
        f_MessageSet(_stMsg);
      END_IF
    END_IF

  //-----------------------------------------------------------------------------------------------
  //-----------------------------------------------------------------------------------------------
  INIT_NCT_BASE_UNIT_COUNT:
    _nNctBaseUnitCount              := TO_UINT(_fbNctController.GetBaseUnitInterfaceCount());

    IF NOT (_nNctBaseUnitCount > 0)
    THEN
      _eState                       := E_PROGRESS.PROGRESS_OCCUPIED;

      IF (_eMessageLevel = E_MessageType.eMessageVerbose)
      THEN
        _stMsg.eType                := E_MessageType.eMessageVerbose;
        _stMsg.eSubdevice           := e_Subdevice.Xpu_fbNctBaseUnit;
        _stMsg.iErrorNumber         := 0;
        _stMsg.sText                := concat(TO_STRING(_eState), ': ');
        _stMsg.sText                := concat(_stMsg.sText, TO_STRING(_nState));
        f_MessageSet(_stMsg);
      END_IF
    ELSE
      _nNctBaseUnitIdx              := 1;
      _nState                       := INIT_NCT_BASE_UNIT_ITF;

      IF (_eMessageLevel = E_MessageType.eMessageVerbose)
      THEN
        _stMsg.eType                := E_MessageType.eMessageVerbose;
        _stMsg.eSubdevice           := e_Subdevice.Xpu_fbNctBaseUnit;
        _stMsg.iErrorNumber         := _nNctBaseUnitCount;
        _stMsg.sText                := concat(TO_STRING(_eState), ': ');
        _stMsg.sText                := concat(_stMsg.sText, TO_STRING(_nState));
        f_MessageSet(_stMsg);
      END_IF
    END_IF

  //-----------------------------------------------------------------------------------------------
  //-----------------------------------------------------------------------------------------------
  INIT_NCT_BASE_UNIT_ITF:
    _ItfNctBaseUnit[_nNctBaseUnitIdx] := _fbNctController.BaseUnitInterfaceTcIo(_nNctBaseUnitIdx);
    _nState                           := INIT_NCT_BASE_UNIT_NEXT;

  //-----------------------------------------------------------------------------------------------
  //-----------------------------------------------------------------------------------------------
  INIT_NCT_BASE_UNIT_NEXT:
    IF (_nNctBaseUnitIdx > _nNctBaseUnitCount-1)
    THEN
      _eState                       := E_PROGRESS.PROGRESS_OCCUPIED;
    ELSE
      _nNctBaseUnitIdx              := _nNctBaseUnitIdx + 1;
      _nState                       := INIT_NCT_BASE_UNIT_ITF;
    END_IF
  END_CASE
END_CASE
//-----------------------------------------------------------------------------------------------
//-----------------------------------------------------------------------------------------------
//-----------------------------------------------------------------------------------------------
CASE _eState
OF
  E_PROGRESS.PROGRESS_OCCUPIED:     // reserve
    _eState                         := E_PROGRESS.PROGRESS_WORKING;
END_CASE
//-----------------------------------------------------------------------------------------------
//-----------------------------------------------------------------------------------------------
//-----------------------------------------------------------------------------------------------
CASE _eState
OF
  E_PROGRESS.PROGRESS_WORKING:      // reserve
    _eState                         := E_PROGRESS.PROGRESS_STILL_WORKING;
    _nState                         := INIT_TRACK_COM;
END_CASE
//-----------------------------------------------------------------------------------------------
//-----------------------------------------------------------------------------------------------
//-----------------------------------------------------------------------------------------------
CASE _eState
OF
  E_PROGRESS.PROGRESS_STILL_WORKING:// connect local instances of track, part, modules and mover
  CASE _nState
  OF
  //-----------------------------------------------------------------------------------------------
  //-----------------------------------------------------------------------------------------------
  INIT_TRACK_COM:                   // get TcCom Object for my track (_nTrack is fixed to 1 in this example; multi track is not intended)
    IF _fbXpuTrack.GetComObject(_Track_OTCID[_nTrack])
    THEN
      _nState                       := INIT_PART_COM;

      IF (_eMessageLevel = E_MessageType.eMessageVerbose)
      THEN
        _stMsg.eType                := E_MessageType.eMessageVerbose;
        _stMsg.eSubdevice           := e_Subdevice.Xpu_fbXpuTrack;
        _stMsg.iErrorNumber         := _nTrack;
        _stMsg.sText                := concat(TO_STRING(_eState), ': ');
        _stMsg.sText                := concat(_stMsg.sText, TO_STRING(_nState));
        f_MessageSet(_stMsg);
      END_IF
    END_IF
  //-----------------------------------------------------------------------------------------------
  //-----------------------------------------------------------------------------------------------
  INIT_PART_COM:                    // get TcCom object for my part (also fixed to 1 part per ProcessingUnit; multi part is not intended)
    IF _fbXpuPart.GetComObject(_Part_OTCID[1])
    THEN
      _nState                       := INIT_PART_MODULE_COUNT;

      IF (_eMessageLevel = E_MessageType.eMessageVerbose)
      THEN
        _stMsg.eType                := E_MessageType.eMessageVerbose;
        _stMsg.eSubdevice           := e_Subdevice.Xpu_fbXpuPart;
        _stMsg.iErrorNumber         := 1;
        _stMsg.sText                := concat(TO_STRING(_eState), ': ');
        _stMsg.sText                := concat(_stMsg.sText, TO_STRING(_nState));
        f_MessageSet(_stMsg);
      END_IF
    END_IF
  //-----------------------------------------------------------------------------------------------
  //-----------------------------------------------------------------------------------------------
  INIT_PART_MODULE_COUNT:           // get count of motor modules
    _nModuleCount                   := TO_UINT(_fbXpuPart.GetModuleCount());
  
    IF (_nModuleCount > 0)          // one is enough
    THEN
      _nState                       := INIT_PART_MODULE_OID;

      IF (_eMessageLevel = E_MessageType.eMessageVerbose)
      THEN
        _stMsg.eType                := E_MessageType.eMessageVerbose;
        _stMsg.eSubdevice           := e_Subdevice.Xpu_fbXpuPart;
        _stMsg.iErrorNumber         := _nModuleCount;
        _stMsg.sText                := concat(TO_STRING(_eState), ': ');
        _stMsg.sText                := concat(_stMsg.sText, TO_STRING(_nState));
        f_MessageSet(_stMsg);
      END_IF
    END_IF
  //-----------------------------------------------------------------------------------------------
  //-----------------------------------------------------------------------------------------------
  INIT_PART_MODULE_OID:             // get object IDs of all motor modules in part
    IF _fbXpuPart.GetModuleOids()
    THEN
      _Module_OTCID                 := _fbXpuPart.P_ModuleOids; // copy IDs to local
  
      _nState                       := INIT_PART_MODULE_COM;    // go, connect module IDs
      _nModuleIdx                   := 1;                       // start at first module

      IF (_eMessageLevel = E_MessageType.eMessageVerbose)
      THEN
        _stMsg.eType                := E_MessageType.eMessageVerbose;
        _stMsg.eSubdevice           := e_Subdevice.Xpu_fbPartModules;
        _stMsg.iErrorNumber         := _nModuleIdx;
        _stMsg.sText                := concat(TO_STRING(_eState), ': ');
        _stMsg.sText                := concat(_stMsg.sText, TO_STRING(_nState));
        //f_MessageSet(_stMsg);
      END_IF
    END_IF
  //-----------------------------------------------------------------------------------------------
  //-----------------------------------------------------------------------------------------------
  INIT_PART_MODULE_COM:           // connect to TcCom object
    IF _fbPartModules[_nModuleIdx].GetComObject(_Module_OTCID[_nModuleIdx])
    THEN
      _nState                       := INIT_PART_MODULE_COM_NEXT;
    END_IF
  //-----------------------------------------------------------------------------------------------
  INIT_PART_MODULE_COM_NEXT:
    IF (_nModuleIdx > _nModuleCount-1)
    THEN
      // all data from modules collected, continue to mover data
      _nState                       := INIT_MOVER_COM;          // go, connect mover IDs 
      _nMoverIdx                    :=  1;                      // start at first mover

      IF (_eMessageLevel = E_MessageType.eMessageVerbose)
      THEN
        _stMsg.eType                := E_MessageType.eMessageVerbose;
        _stMsg.eSubdevice           := e_Subdevice.Xpu_fbMoverXpu;
        _stMsg.iErrorNumber         := _nMoverIdx;
        _stMsg.sText                := concat(TO_STRING(_eState), ': ');
        _stMsg.sText                := concat(_stMsg.sText, TO_STRING(_nState));
        //f_MessageSet(_stMsg);
      END_IF
    ELSE
      // still data to fetch, increment search index, go back to fetching data
      _nState                       := INIT_PART_MODULE_COM;    // go back for next
      _nModuleIdx                   := _nModuleIdx + 1;       // next

      IF (_eMessageLevel = E_MessageType.eMessageVerbose)
      THEN
        _stMsg.eType                := E_MessageType.eMessageVerbose;
        _stMsg.eSubdevice           := e_Subdevice.Xpu_fbPartModules;
        _stMsg.iErrorNumber         := _nModuleIdx;
        _stMsg.sText                := concat(TO_STRING(_eState), ': ');
        _stMsg.sText                := concat(_stMsg.sText, TO_STRING(_nState));
        //f_MessageSet(_stMsg);
      END_IF
    END_IF
  //-----------------------------------------------------------------------------------------------
  //-----------------------------------------------------------------------------------------------
  INIT_MOVER_COM:                   // connect to TcCom object
    IF _fbMoverXpu[_nMoverIdx].GetComObject(_Mov_OTCID[_nMoverIdx])
    THEN
      _nState                       := INIT_MOVER_COM_NEXT;
    END_IF
  //-----------------------------------------------------------------------------------------------
  INIT_MOVER_COM_NEXT:
    IF (_nMoverIdx > _nMoverCount-1)
    THEN
      // all done
      _nState                       := INIT_DATA_GET;           // get important data from ProcessingUnit etc...

      IF (_eMessageLevel = E_MessageType.eMessageVerbose)
      THEN
        _stMsg.eType                := E_MessageType.eMessageVerbose;
        _stMsg.eSubdevice           := e_Subdevice.Xpu_fbProcessingUnit;
        _stMsg.iErrorNumber         := 0;
        _stMsg.sText                := concat(TO_STRING(_eState), ': ');
        _stMsg.sText                := concat(_stMsg.sText, TO_STRING(_nState));
        f_MessageSet(_stMsg);
      END_IF
    ELSE
      // more data to fetch, increment search index and go back
      _nState                       := INIT_MOVER_COM;          // go back for next
      _nMoverIdx                    := _nMoverIdx + 1;       // next

      IF (_eMessageLevel = E_MessageType.eMessageVerbose)
      THEN
        _stMsg.eType                := E_MessageType.eMessageVerbose;
        _stMsg.eSubdevice           := e_Subdevice.Xpu_fbMoverXpu;
        _stMsg.iErrorNumber         := _nMoverIdx;
        _stMsg.sText                := concat(TO_STRING(_eState), ': ');
        _stMsg.sText                := concat(_stMsg.sText, TO_STRING(_nState));
        //f_MessageSet(_stMsg);
      END_IF
    END_IF
  //-----------------------------------------------------------------------------------------------
  //-----------------------------------------------------------------------------------------------
  INIT_DATA_GET:                    // get data, add more if your application requires it
    // start counter
    _eDataGetCount                  := _eDataGetCount + 1;
    IF (_eDataGetCount MOD E_PROGRESS.PROGRESS_ERROR = 0)
    THEN
      _eState                       := E_PROGRESS.PROGRESS_ERROR;
      _eCheck                       := E_XPU_CHECK.PROCESSING_UNIT_GET_DATA_EXCEED;

      _stMsg.eType                  := E_MessageType.eMessageError;
      _stMsg.eSubdevice             := e_Subdevice.Xpu_fbProcessingUnit;
      _stMsg.iErrorNumber           := _nMoverIdx;
      _stMsg.sText                  := concat(TO_STRING(_nState), ': ');
      _stMsg.sText                  := concat(_stMsg.sText, TO_STRING(_eCheck));
      f_MessageSet(_stMsg);
    END_IF
    // wait for plausible data from members
    IF (_bAllPositionsValid) AND
       (_nLengthXpu > 0)
    THEN
      _nState                       := INIT_DATA_CHECK;
      _eChk                         := E_XPU_CHECK.PROCESSING_UNIT_POSITIONS_VALID;
      IF (_eMessageLevel > E_MessageType.eMessageError)
      THEN
        _stMsg.eType                := E_MessageType.eMessageInfo;
        _stMsg.eSubdevice           := e_Subdevice.Xpu_fbProcessingUnit;
        _stMsg.iErrorNumber         := 0;
        _stMsg.sText                := concat(TO_STRING(_nState), ': ');
        _stMsg.sText                := concat(_stMsg.sText, TO_STRING(E_XPU_CHECK.PROCESSING_UNIT_POSITIONS_VALID));
        f_MessageSet(_stMsg);
      END_IF
    END_IF

    _bAllPositionsValid             := _fbProcessingUnit.GetAreAllPositionsValid();
    _nDetectedMoverCount            := TO_UINT(_fbProcessingUnit.GetDetectedMoverCount());
    _nExpectedMoverCount            := TO_UINT(_fbProcessingUnit.GetExpectedMoverCount());

    _XpuOperationMode               := _fbProcessingUnit.GetOperationMode();
    _MoverIdDetectionMode           := _fbProcessingUnit.GetMoverIdDetectionMode();

    _RailLengthXpu                  := _fbXpuPart.GetLength();
    _RailLengthGroup                := _fbMc2CaGroup.GetRailLength();
    _nLengthXpu                     := TO_UINT(_RailLengthXpu);
    _nLengthGroup                   := TO_UINT(_RailLengthGroup);

  //-----------------------------------------------------------------------------------------------
  //-----------------------------------------------------------------------------------------------
  INIT_DATA_CHECK:                  // plausibility checks
    IF NOT (_nDetectedMoverCount = _nExpectedMoverCount)
    THEN
      _eChk                         := E_XPU_CHECK.MOVER_COUNT_NOT_EQUAL; // the thing that must not be
      _eState                       := E_PROGRESS.PROGRESS_ERROR;

      _stMsg.eType                  := E_MessageType.eMessageError;
      _stMsg.eSubdevice             := e_Subdevice.Xpu_fbProcessingUnit;
      _stMsg.iErrorNumber           := _nMoverIdx;
      _stMsg.sText                  := concat(TO_STRING(_nState), ': ');
      _stMsg.sText                  := concat(_stMsg.sText, TO_STRING(E_XPU_CHECK.MOVER_COUNT_NOT_EQUAL));
      f_MessageSet(_stMsg);

    ELSIF NOT (_nLengthXpu = _nLengthGroup)
    THEN
      _eChk                         := E_XPU_CHECK.RAIL_LENGTH_COMPARE;   // yet another thing that must not be
      _eState                       := E_PROGRESS.PROGRESS_ERROR;

      _stMsg.eType                  := E_MessageType.eMessageError;
      _stMsg.eSubdevice             := e_Subdevice.Xpu_fbProcessingUnit;
      _stMsg.iErrorNumber           := _nMoverIdx;
      _stMsg.sText                  := concat(TO_STRING(_nState), ': ');
      _stMsg.sText                  := concat(_stMsg.sText, TO_STRING(E_XPU_CHECK.RAIL_LENGTH_COMPARE));
      f_MessageSet(_stMsg);
    ELSE
      _sVersionXpu                  := _fbProcessingUnit.GetVersionString();
      _nState                       := INIT_DONE;                         // write success
    END_IF

  //-----------------------------------------------------------------------------------------------
  //-----------------------------------------------------------------------------------------------
  INIT_DONE:
    _eState                         := E_PROGRESS.PROGRESS_DONE;          // method is done
    IF (_eMessageLevel > E_MessageType.eMessageError)
    THEN
      _stMsg.eType                  := E_MessageType.eMessageInfo;
      _stMsg.eSubdevice             := e_Subdevice.Xpu_fbProcessingUnit;
      _stMsg.iErrorNumber           := 0;
      _stMsg.sText                  := concat('Xpu VersionString: ', _sVersionXpu);
      f_MessageSet(_stMsg);

      _stMsg.eType                  := E_MessageType.eMessageInfo;
      _stMsg.eSubdevice             := e_Subdevice.Xpu_fbProcessingUnit;
      _stMsg.iErrorNumber           := 0;
      _stMsg.sText                  := concat(TO_STRING(_nState), ': ');
      _stMsg.sText                  := concat(_stMsg.sText, TO_STRING(_eState));
      f_MessageSet(_stMsg);
    END_IF
  END_CASE
END_CASE
//-----------------------------------------------------------------------------------------------
//-----------------------------------------------------------------------------------------------
//-----------------------------------------------------------------------------------------------
_eReslt                             := _eState;
XpuInit                             := _nState;
//-----------------------------------------------------------------------------------------------
//-----------------------------------------------------------------------------------------------
//-----------------------------------------------------------------------------------------------
END_METHOD

PROPERTY XpuInstance : uint
SET
//
// Who am I?
// Environment may have more than one ProcessingUnit,
// information required for connecting to the correct instance of ProcessingUnit
_nXpu := XpuInstance;
END_SET
END_PROPERTY

PROPERTY XpuModuleInfoData : REFERENCE TO ARRAY[1..MAX_MODULE] OF Tc3_XTS_Utility.ST_InfoDataView
SET

_ModuleInfoData REF= XpuModuleInfoData;
END_SET
END_PROPERTY

PROPERTY XpuOtcid : OTCID
GET
XpuOtcid := _Xpu_OTCID;
END_GET
END_PROPERTY

END_FUNCTION_BLOCK

// ---- APPLICATION/_Visu/SIM_TEST.TcVIS
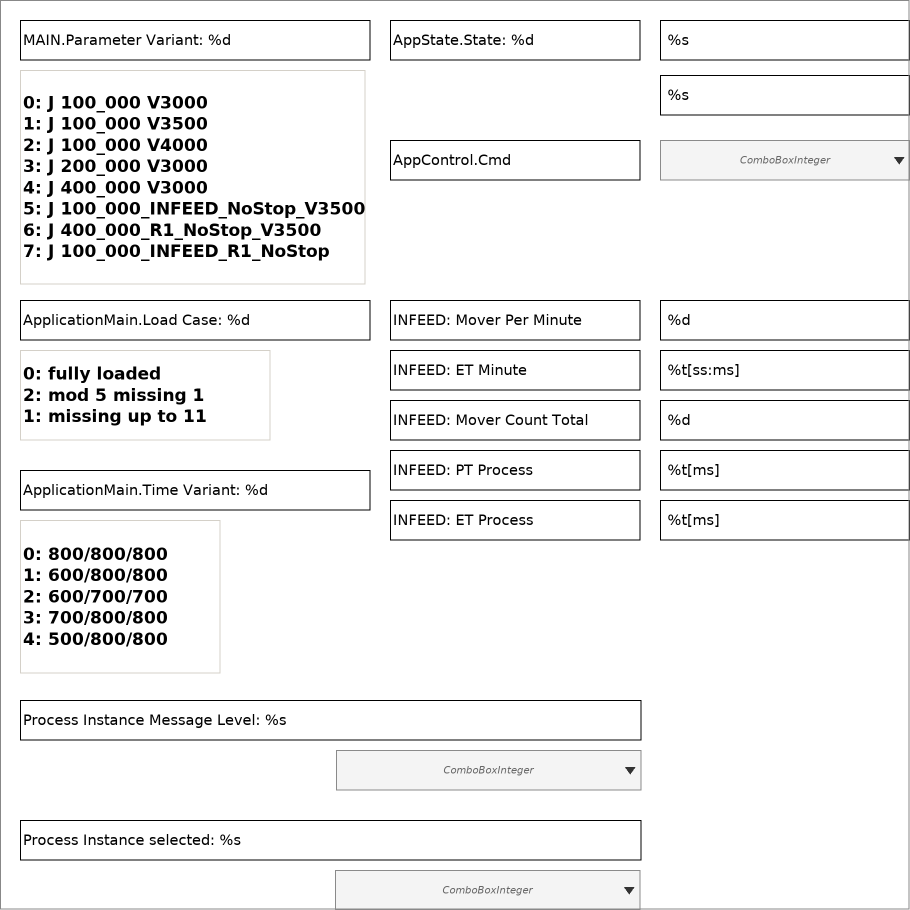
VISUALIZATION SIM_TEST  // 910x910
    Rectangle (20,300 350x40), "ApplicationMain.Load Case: %d", text variable: GVL_APPLICATION.ApplicationMain._nLoadCase
        OnMouseClick: write the text variable via VisuDialogs.Numpad, min 0, max 2
    Rectangle (20,470 350x40), "ApplicationMain.Time Variant: %d", text variable: GVL_APPLICATION.ApplicationMain._nTimeVariant
        OnMouseClick: write the text variable via VisuDialogs.Numpad, min 0, max 100
    Rectangle (20,20 350x40), "MAIN.Parameter Variant: %d", text variable: MAIN.nParameterVariant
        OnMouseClick: write the text variable via VisuDialogs.Numpad, min 0, max 100
    Textfield (20,520 200x153), "0: 800/800/800 1: 600/800/800 2: 600/700/700 3: 700/800/800 4: 500/800/800"
    Textfield (20,350 250x90), "0: fully loaded 2: mod 5 missing 1 1: missing up to 11"
    Textfield (20,70 345x214), "0: J 100_000 V3000 1: J 100_000 V3500 2: J 100_000 V4000 3: J 200_000 V3000 4: J 400_000 V3000 5: J 100_000_INFEED_NoStop_V3500 6: J 400_000_R1_NoStop_V3500 7: J 100_000_INFEED_R1_NoStop"
    Rectangle (390,140 250x40), "AppControl.Cmd"
    ComboBoxInteger (660,140 250x40), variable: GVL_APPLICATION.AppControl.Cmd, text list: 'TL_E_INSTANCE_CMD'
    Rectangle (390,20 250x40), "AppState.State: %d", text variable: GVL_APPLICATION.AppState.AppState
    Rectangle (660,75 250x40), "%s", text variable: GVL_APPLICATION.ApplicationMain._sAppResult
    Rectangle (390,300 250x40), "INFEED: Mover Per Minute"
    Rectangle (660,300 250x40), "%d", text variable: GVL_APPLICATION.ProcessCollector[2]._AllStationMoverPerMinute
    Rectangle (390,400 250x40), "INFEED: Mover Count Total"
    Rectangle (660,400 250x40), "%d", text variable: GVL_APPLICATION.ProcessCollector[2]._nMoverCountTotal
    Rectangle (390,500 250x40), "INFEED: ET Process"
    Rectangle (660,500 250x40), "%t[ms]", text variable: GVL_APPLICATION.ApplicationMain._tonProcess[2].ET
    Rectangle (390,450 250x40), "INFEED: PT Process"
    Rectangle (660,450 250x40), "%t[ms]", text variable: GVL_APPLICATION.ApplicationMain._tProcess[2]
    Rectangle (390,350 250x40), "INFEED: ET Minute"
    Rectangle (660,350 250x40), "%t[ss:ms]", text variable: ProcessCollector[2]._tonPartsPerMinute.ET
    Rectangle (660,20 250x40), "%s", text variable: GVL_APPLICATION.ApplicationMain._sAppState
    Rectangle (20,700 621x40), "Process Instance Message Level: %s", text variable: MessageData.sMessageLevelSelected
    ComboBoxInteger (335,870 305x40), variable: MessageData.nProcessSelected, text list: 'TL_E_INSTANCE'
    ComboBoxInteger (336,750 305x40), variable: GVL_MSG.MessageLevelProcess[MessageData.nProcessSelected], text list: 'TL_E_MESSAGETYPE'
    Rectangle (20,820 621x40), "Process Instance selected: %s", text variable: MessageData.sProcessSelected
END_VISUALIZATION

// ---- APPLICATION/_Visu/textlists/TL_E_INSTANCE.TcTLO
TEXTLIST TL_E_INSTANCE
  1 = 'BUFFER_INFEED'
  2 = 'INFEED'
  3 = 'BUFFER_OUTFEED_ROBOT'
  4 = 'OUTFEED_ROBOT_R1'
  5 = 'OUTFEED_ROBOT_R2'
  6 = 'SENDER_FAST'
  7 = 'SENDER_BUFFER_INFEED'
   = ''
END_TEXTLIST

// ---- GlobalTextList.TcGTLO
TEXTLIST GlobalTextList
  161 = ' %d'
  781 = ' %s'
  290 = ' %t[ms]'
  1009 = ' %t[ss:ms]'
  17 = ' STATION_ENABLE'
  34 = ' STATION_MOVER_ENTER'
  452 = ' STATION_MOVER_GONE'
  75 = ' STATION_MOVER_OUT'
  598 = ' STATION_PROCESS_DONE'
  750 = ' STATION_PROCESS_START'
  294 = '%.2f'
  191 = '%d'
  836 = '%s'
  1246 = '0: 800/800/800\n1: 600/800/800\n2: 600/700/700\n3: 700/800/800\n4: 500/800/800'
  605 = '0: fully loaded\n2: mod 5 missing 1\n1: missing up to 11'
  1159 = '0: J 100_000 V3000\n1: J 100_000 V3500\n2: J 100_000 V4000\n3: J 200_000 V3000\n4: J 400_000 V3000\n5: J 100_000 PosStop 0.0 V3500'
  666 = '0: J 100_000 V3000\n1: J 100_000 V3500\n2: J 100_000 V4000\n3: J 200_000 V3000\n4: J 400_000 V3000\n5: J 100_000 PosStop 0.0 V3500\n6: J_400_000_R1_NoStop_V3500'
  699 = '0: J 100_000 V3000\n1: J 100_000 V3500\n2: J 100_000 V4000\n3: J 200_000 V3000\n4: J 400_000 V3000\n5: J 100_000_INFEED_NoStop_V3500\n6: J 400_000_R1_NoStop_V3500'
  510 = '0: J 100_000 V3000\n1: J 100_000 V3500\n2: J 100_000 V4000\n3: J 200_000 V3000\n4: J 400_000 V3000\n5: J 100_000_INFEED_NoStop_V3500\n6: J 400_000_R1_NoStop_V3500\n7: J 100_000_INFEED_R1_NoStop'
  248 = 'Activate'
  444 = 'Activate Visu list'
  704 = 'All Positions Valid'
  562 = 'AllAxisStanding'
  667 = 'AppControl.Cmd'
  32 = 'ApplicationMain.Load Case: %d'
  459 = 'ApplicationMain.Time Variant: %d'
  295 = 'AppState.State'
  906 = 'AppState.State: %d'
  878 = 'AxisCount Enabled: %d'
  162 = 'AxisCount: %d'
  914 = 'ConstantVelocity'
  929 = 'Control'
  707 = 'CyclicCheck: %s'
  660 = 'DC Link All Modules'
  359 = 'Decelerating'
  843 = 'Detected AxisCount: %d'
  243 = 'eDevice'
  244 = 'eSubdevice'
  242 = 'eType'
  772 = 'Expected AxisCount: %d'
  48 = 'GroupDisabled'
  915 = 'GroupError'
  495 = 'GroupErrorId: %d'
  975 = 'GroupErrorStop'
  940 = 'GroupHoming'
  300 = 'GroupMoving'
  807 = 'GroupNotReady'
  438 = 'GroupStandby'
  226 = 'GroupStatusBusy'
  204 = 'GroupStatusValid'
  973 = 'GroupStopping'
  942 = 'GVL_XTS.CaGroupInfo'
  680 = 'ID Detection Active'
  238 = 'ID Detection Error'
  526 = 'ID Detection Mode: %s'
  29 = 'ID Detection Valid'
  245 = 'iErrorNumber'
  358 = 'INFEED: ET Minute'
  328 = 'INFEED: ET Process'
  268 = 'INFEED: Mover Count Total'
  682 = 'INFEED: Mover Per Minute'
  928 = 'INFEED: PT Process'
  211 = 'Info Act Pos Absolute'
  586 = 'Info Act Pos Modulo'
  21 = 'Info Mover Avoiding Collision'
  282 = 'Info Mover Coupled'
  398 = 'Info Mover Enabled'
  751 = 'Info Mover Error'
  907 = 'Info Mover Standstill'
  480 = 'Info nError ID'
  922 = 'Info Target Pos Absolute'
  16 = 'Info Target Pos Modulo'
  616 = 'InPosition'
  356 = 'MAIN.Parameter Variant: %d'
  713 = 'Mask: %b'
  972 = 'Mask: %d'
  779 = 'Mask: %s'
  726 = 'McGroupState:      %s'
  160 = 'McGroupState: %d  %s'
  974 = 'MOVER command'
  387 = 'Mover ID: %d'
  297 = 'Mover Position Assignement: %s'
  840 = 'MOVER result:  %s'
  53 = 'MOVER state:   %s'
  756 = 'nMoverSelected: %d'
  669 = 'nStation selected: %d'
  94 = 'Offset %.3f'
  427 = 'Offset: %.3f'
  312 = 'Operation Mode: %s'
  140 = 'Process Instance Message Level: %s'
  899 = 'Process Instance selected: %s'
  1106 = 'Process Instances Message Level: %d'
  178 = 'Process Instances Message Level: %s'
  369 = 'Process Instances Message Level: %s; %s'
  205 = 'Process Instances selected: %s'
  320 = 'Queue: %d'
  91 = 'Set Acceleration'
  399 = 'Set Delta'
  382 = 'Set Distance'
  757 = 'Set Gap'
  934 = 'Set Jerk'
  201 = 'Set Override'
  936 = 'Set Position'
  62 = 'Set Velocity'
  231 = 'State'
  748 = 'Station Control'
  267 = 'Station State'
  627 = 'STATION_ENABLE'
  247 = 'sText'
  54 = 'Target Station %d'
  567 = 'Target Station: %d'
  246 = 'tTime'
  517 = 'WRITE TO FILE'
  275 = 'XPU Command'
  227 = 'XpuResult:   %s'
  96 = 'XpuState:    %s'
  884 = 'XTS Station'
  572 = 'XTS Transport Check:  %s'
  212 = 'XTS Transport Check: %s'
  500 = 'XTS Transport Command'
  395 = 'XTS Transport Result: %s'
  798 = 'XTS Transport State:  %s'
  417 = 'XTS Transport State: %s'
END_TEXTLIST

// ---- MSG/T_MESSAGE_LIST.TcVIS
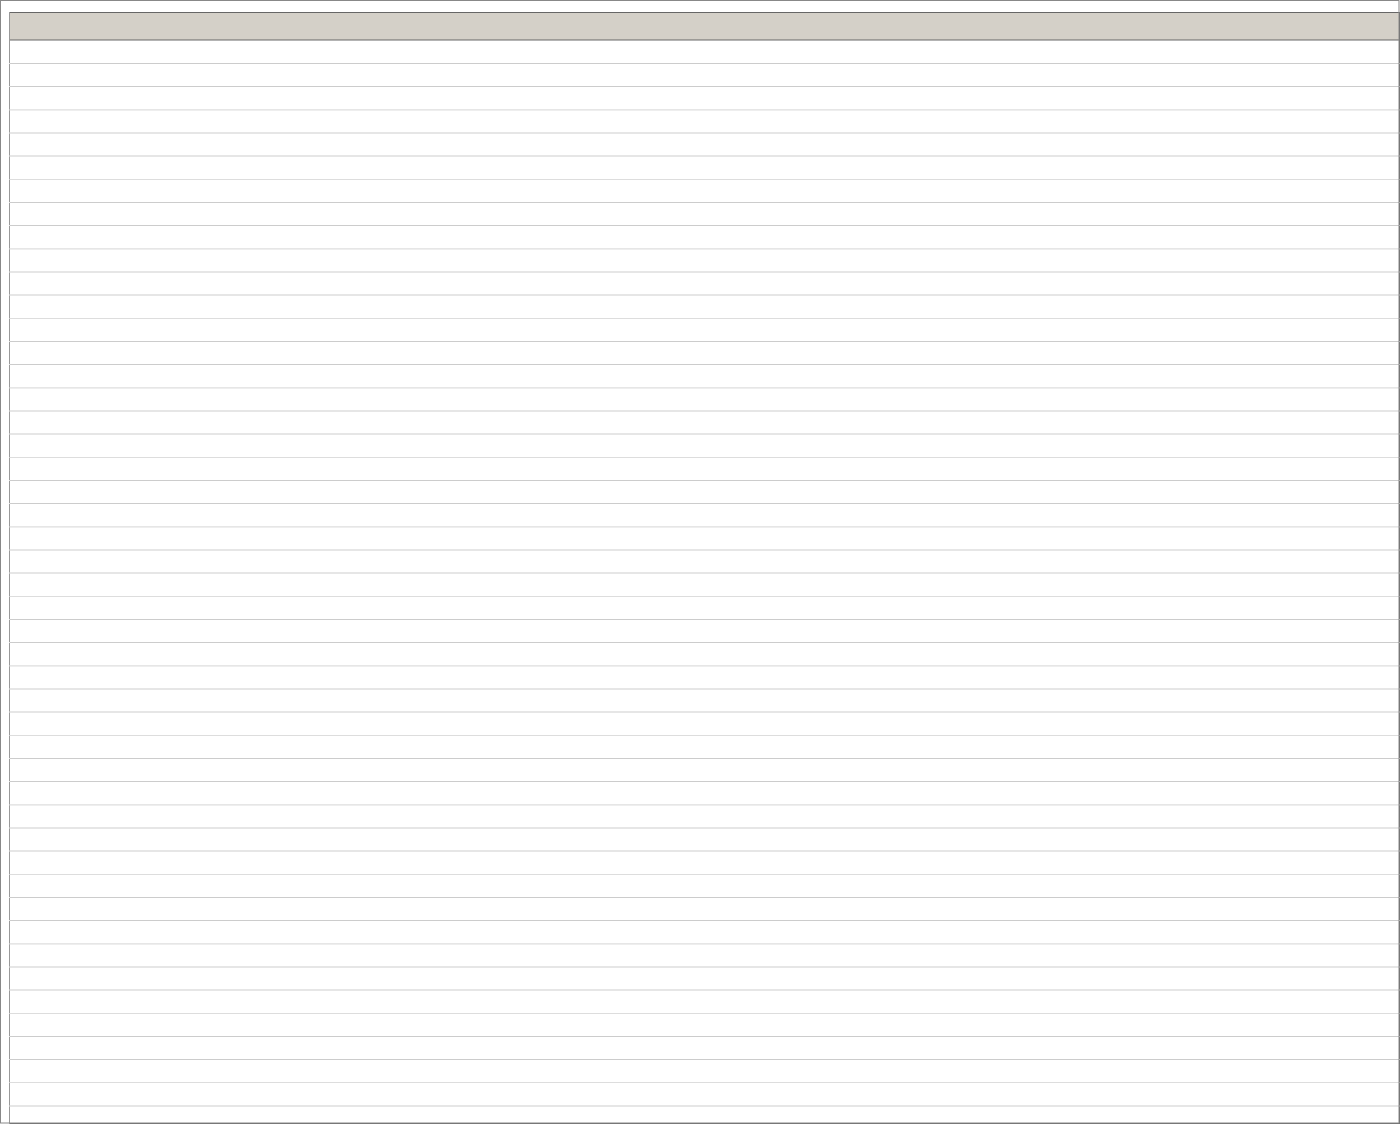
VISUALIZATION T_MESSAGE_LIST  // 1510x1213
    Table (10,13 1500x1200), data array: MessageData.VisuList
        p1128707560: GVL_AXIS_CTRL.MAX_MESSAGE
        p3854506369: MessageData.VisuList[INDEX].eType
        p1892666644: MessageData.VisuList[INDEX].eDevice
        p338671338: MessageData.VisuList[INDEX].eSubdevice
        p2170511999: MessageData.VisuList[INDEX].iErrorNumber
        p3723444502: MessageData.VisuList[INDEX].tTime
        p1218418051: MessageData.VisuList[INDEX].sText
END_VISUALIZATION

// ---- XTS/_Visualization/GROUP_VISU.TcVIS
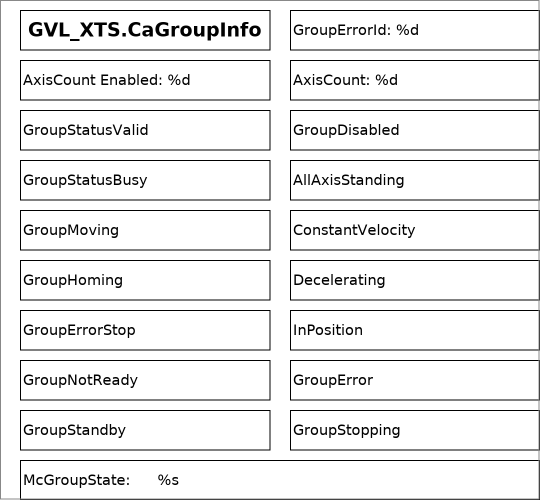
VISUALIZATION GROUP_VISU  // 540x500
    Rectangle (20,110 250x40), "GroupStatusValid", colour toggle: GVL_XTS.XtsTransportState.GroupInfo.GroupStatusValid
    Rectangle (20,160 250x40), "GroupStatusBusy", colour toggle: GVL_XTS.XtsTransportState.GroupInfo.GroupStatusBusy
    Rectangle (20,210 250x40), "GroupMoving", colour toggle: GVL_XTS.XtsTransportState.GroupInfo.GroupMoving
    Rectangle (20,260 250x40), "GroupHoming", colour toggle: GVL_XTS.XtsTransportState.GroupInfo.GroupHoming
    Rectangle (20,310 250x40), "GroupErrorStop", colour toggle: GVL_XTS.XtsTransportState.GroupInfo.GroupErrorStop
    Rectangle (20,360 250x40), "GroupNotReady", colour toggle: GVL_XTS.XtsTransportState.GroupInfo.GroupNotReady
    Rectangle (20,410 250x40), "GroupStandby", colour toggle: GVL_XTS.XtsTransportState.GroupInfo.GroupStandby
    Rectangle (290,410 250x40), "GroupStopping", colour toggle: GVL_XTS.XtsTransportState.GroupInfo.GroupStopping
    Rectangle (290,110 250x40), "GroupDisabled", colour toggle: GVL_XTS.XtsTransportState.GroupInfo.GroupDisabled
    Rectangle (290,160 250x40), "AllAxisStanding", colour toggle: GVL_XTS.XtsTransportState.GroupInfo.AllAxesStanding
    Rectangle (290,210 250x40), "ConstantVelocity", colour toggle: GVL_XTS.XtsTransportState.GroupInfo.ConstantVelocity
    Rectangle (290,260 250x40), "Decelerating", colour toggle: GVL_XTS.XtsTransportState.GroupInfo.Decelerating
    Rectangle (290,310 250x40), "InPosition", colour toggle: GVL_XTS.XtsTransportState.GroupInfo.InPosition
    Rectangle (290,360 250x40), "GroupError", colour toggle: GVL_XTS.XtsTransportState.GroupInfo.GroupError
    Rectangle (290,10 250x40), "GroupErrorId: %d", text variable: GVL_XTS.XtsTransportState.GroupInfo.GroupErrorId
    Rectangle (290,60 250x40), "AxisCount: %d", text variable: GVL_XTS.XtsTransportState.GroupInfo.AxisCount
    Rectangle (20,460 520x40), "McGroupState: %s", text variable: MAIN.sCaGroupState
    Rectangle (20,10 250x40), "GVL_XTS.CaGroupInfo"
    Rectangle (20,60 250x40), "AxisCount Enabled: %d", text variable: GVL_XTS.CaGroupInfo.AxisCountEnabled
END_VISUALIZATION

// ---- XTS/_Visualization/MOVER_VISU.TcVIS
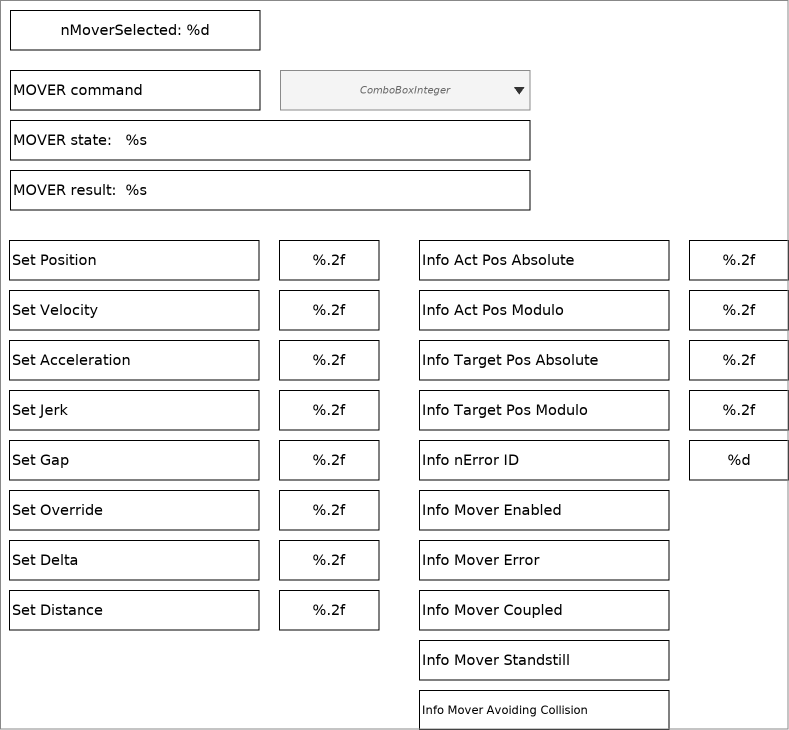
VISUALIZATION MOVER_VISU  // 789x730
    Rectangle (10,10 250x40), "nMoverSelected: %d", text variable: MAIN.nMoverSelected
        OnMouseClick: write the text variable via VisuDialogs.Numpad, min 1, max MAX_MOVER, title 'Selected Mover'
    Rectangle (10,120 520x40), "MOVER state: %s", text variable: MAIN.sMoverState
    Rectangle (10,70 250x40), "MOVER command"
    ComboBoxInteger (280,70 250x40), variable: GVL_XTS.MoverCtrl[MAIN.nMoverSelected].Cmd, text list: 'TL_E_CTRL_MOVER'
    Rectangle (10,170 520x40), "MOVER result: %s", text variable: MAIN.sMoverResult
    Rectangle (9,240 250x40), "Set Position"
    Rectangle (9,290 250x40), "Set Velocity"
    Rectangle (9,340 250x40), "Set Acceleration"
    Rectangle (9,390 250x40), "Set Jerk"
    Rectangle (9,440 250x40), "Set Gap"
    Rectangle (9,490 250x40), "Set Override"
    Rectangle (9,540 250x40), "Set Delta"
    Rectangle (9,590 250x40), "Set Distance"
    Rectangle (279,240 100x40), "%.2f", text variable: GVL_XTS.MoveData[MAIN.nMoverSelected].rPos
        OnMouseClick: write the text variable via Default
    Rectangle (279,290 100x40), "%.2f", text variable: GVL_XTS.MoveData[MAIN.nMoverSelected].rVelo
        OnMouseClick: write the text variable via Default
    Rectangle (279,340 100x40), "%.2f", text variable: GVL_XTS.MoveData[MAIN.nMoverSelected].rAcc
        OnMouseClick: write the text variable via Default
    Rectangle (279,390 100x40), "%.2f", text variable: GVL_XTS.MoveData[MAIN.nMoverSelected].rJerk
        OnMouseClick: write the text variable via Default
    Rectangle (279,440 100x40), "%.2f", text variable: GVL_XTS.MoveData[MAIN.nMoverSelected].rGap
        OnMouseClick: write the text variable via Default
    Rectangle (279,490 100x40), "%.2f", text variable: GVL_XTS.MoveData[MAIN.nMoverSelected].rOverride
        OnMouseClick: write the text variable via Default
    Rectangle (279,540 100x40), "%.2f", text variable: GVL_XTS.MoveData[MAIN.nMoverSelected].rDelta
        OnMouseClick: write the text variable via Default
    Rectangle (279,590 100x40), "%.2f", text variable: GVL_XTS.MoveData[MAIN.nMoverSelected].rDistance
        OnMouseClick: write the text variable via Default
    Rectangle (419,240 250x40), "Info Act Pos Absolute"
    Rectangle (419,290 250x40), "Info Act Pos Modulo"
    Rectangle (419,340 250x40), "Info Target Pos Absolute"
    Rectangle (419,390 250x40), "Info Target Pos Modulo"
    Rectangle (419,440 250x40), "Info nError ID"
    Rectangle (689,240 100x40), "%.2f", text variable: GVL_XTS.MoverInfo[MAIN.nMoverSelected].rAbsActPos
    Rectangle (689,290 100x40), "%.2f", text variable: GVL_XTS.MoverInfo[MAIN.nMoverSelected].rModuloActPos
    Rectangle (689,340 100x40), "%.2f", text variable: GVL_XTS.MoverInfo[MAIN.nMoverSelected].rAbsTargetPos
    Rectangle (689,390 100x40), "%.2f", text variable: GVL_XTS.MoverInfo[MAIN.nMoverSelected].rModuloTargetPos
    Rectangle (689,440 100x40), "%d", text variable: GVL_XTS.MoverInfo[MAIN.nMoverSelected].nErrorId
    Rectangle (419,490 250x40), "Info Mover Enabled", colour toggle: GVL_XTS.MoverInfo[MAIN.nMoverSelected].bMoverEnabled
    Rectangle (419,540 250x40), "Info Mover Error", colour toggle: GVL_XTS.MoverInfo[MAIN.nMoverSelected].bMoverError
    Rectangle (419,590 250x40), "Info Mover Coupled", colour toggle: GVL_XTS.MoverInfo[MAIN.nMoverSelected].bMoverCoupled
    Rectangle (419,640 250x40), "Info Mover Standstill", colour toggle: GVL_XTS.MoverInfo[MAIN.nMoverSelected].bMoverStandstill
    Rectangle (419,690 250x40), "Info Mover Avoiding Collision", colour toggle: GVL_XTS.MoverInfo[MAIN.nMoverSelected].bMoverAvoidingCollision
END_VISUALIZATION

// ---- XTS/_Visualization/STATION_VISU.TcVIS
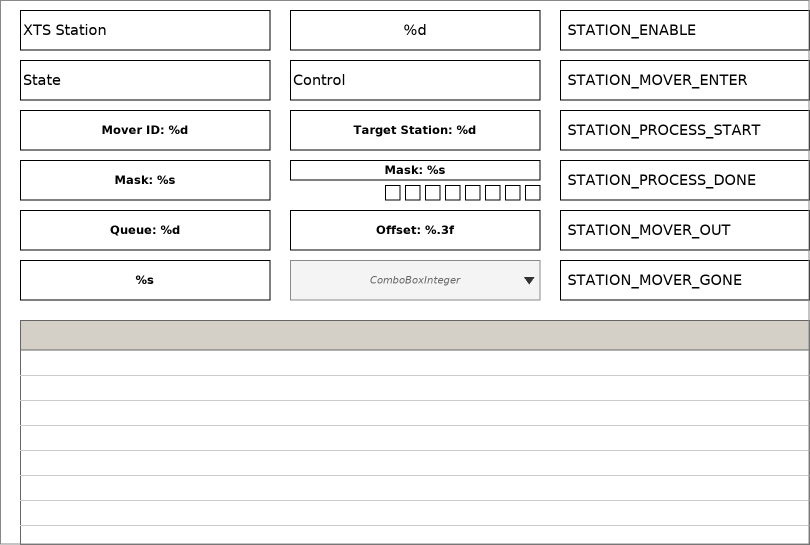
VISUALIZATION STATION_VISU  // 810x545
    Rectangle (20,10 250x40), "XTS Station"
    Rectangle (290,10 250x40), "%d", text variable: MAIN.nStationSelected
        OnMouseClick: write the text variable via VisuDialogs.Numpad, min 1, max MAX_STATION, title 'Selected Station'
    Rectangle (20,60 250x40), "State"
    Rectangle (290,60 250x40), "Control"
    Rectangle (20,210 250x40), "Queue: %d", text variable: GVL_XTS.StationState[MAIN.nStationSelected].nQueue
    Rectangle (20,110 250x40), "Mover ID: %d", text variable: GVL_XTS.StationState[MAIN.nStationSelected].nMoverId
    Rectangle (20,160 250x40), "Mask: %s", text variable: MAIN.sStationStateMask
    Rectangle (20,260 250x40), "%s", text variable: MAIN.sStationState
    ComboBoxInteger (290,260 250x40), variable: GVL_XTS.StationCtrl[MAIN.nStationSelected].eCmd, text list: 'TL_E_CTRL_STATION'
    Rectangle (290,210 250x40), "Offset: %.3f", text variable: GVL_XTS.StationCtrl[MAIN.nStationSelected].rOffset
    Rectangle (290,110 250x40), "Target Station: %d", text variable: GVL_XTS.StationCtrl[MAIN.nStationSelected].nTargetStation
        OnMouseClick: write the text variable via VisuDialogs.Numpad, min 1, max MAX_STATION, title 'Target Station'
    Rectangle (290,160 250x20), "Mask: %s", text variable: MAIN.sStationCtrlMask
    Rectangle (525,185 15x15)
        toggle GVL_XTS.StationCtrl[MAIN.nStationSelected].nMask.0
    Rectangle (505,185 15x15)
        toggle GVL_XTS.StationCtrl[MAIN.nStationSelected].nMask.1
    Rectangle (485,185 15x15)
        toggle GVL_XTS.StationCtrl[MAIN.nStationSelected].nMask.2
    Rectangle (465,185 15x15)
        toggle GVL_XTS.StationCtrl[MAIN.nStationSelected].nMask.3
    Rectangle (445,185 15x15)
        toggle GVL_XTS.StationCtrl[MAIN.nStationSelected].nMask.4
    Rectangle (425,185 15x15)
        toggle GVL_XTS.StationCtrl[MAIN.nStationSelected].nMask.5
    Rectangle (405,185 15x15)
        toggle GVL_XTS.StationCtrl[MAIN.nStationSelected].nMask.6
    Rectangle (385,185 15x15)
        toggle GVL_XTS.StationCtrl[MAIN.nStationSelected].nMask.7
    Rectangle (560,10 250x40), "STATION_ENABLE", colour toggle: MAIN.bStationEnable
        OnMouseClick: execute { GVL_XTS.StationCtrl[MAIN.nStationSelected].eCmd := E_STATION_CTRL.STATION_ENABLE; }
    Rectangle (560,60 250x40), "STATION_MOVER_ENTER", colour toggle: MAIN.bStationEnter
        OnMouseClick: execute { GVL_XTS.StationCtrl[MAIN.nStationSelected].eCmd := E_STATION_CTRL.STATION_MOVER_ENTER; }
    Rectangle (560,110 250x40), "STATION_PROCESS_START", colour toggle: MAIN.bStationStart
        OnMouseClick: execute { GVL_XTS.StationCtrl[MAIN.nStationSelected].eCmd := E_STATION_CTRL.STATION_PROCESS_START; }
    Rectangle (560,160 250x40), "STATION_PROCESS_DONE", colour toggle: MAIN.bStationDone
        OnMouseClick: execute { GVL_XTS.StationCtrl[MAIN.nStationSelected].eCmd := E_STATION_CTRL.STATION_PROCESS_DONE; }
    Rectangle (560,210 250x40), "STATION_MOVER_OUT", colour toggle: MAIN.bStationOut
        OnMouseClick: execute { GVL_XTS.StationCtrl[MAIN.nStationSelected].eCmd := E_STATION_CTRL.STATION_MOVER_OUT; }
    Rectangle (560,260 250x40), "STATION_MOVER_GONE", colour toggle: MAIN.bStationGone
        OnMouseClick: execute { GVL_XTS.StationCtrl[MAIN.nStationSelected].eCmd := E_STATION_CTRL.STATION_MOVER_GONE; }
    Table (20,320 790x225), data array: MAIN.tStationSelectedQueue
        p3854506369: MAIN.tStationSelectedQueue[INDEX].nMoverId
        p1892666644: MAIN.tStationSelectedQueue[INDEX].nTargetStation
        p338671338: MAIN.tStationSelectedQueue[INDEX].nMask
        p2170511999: MAIN.tStationSelectedQueue[INDEX].rOffset
END_VISUALIZATION

// ---- XTS/_Visualization/textlists/TL_E_CTRL_TRANSPORT.TcTLO
TEXTLIST TL_E_CTRL_TRANSPORT
  0 = 'CMD_NULL'
  10 = 'CMD_INIT'
  11 = 'CMD_IDLE'
  20 = 'CMD_MOVER_ENABLE'
  30 = 'CMD_GROUP_CLEAR'
  31 = 'CMD_GROUP_BUILD'
  32 = 'CMD_GROUP_ENABLE'
  40 = 'CMD_TRANSPORT_START'
  41 = 'CMD_TRANSPORT_RESTART'
  21 = 'CMD_MOVER_DISABLE'
  22 = 'CMD_MOVER_HALT_CA'
   = ''
END_TEXTLIST

// ---- XTS/_Visualization/textlists/TL_E_CTRL_XPU.TcTLO
TEXTLIST TL_E_CTRL_XPU
  0 = 'XTS_CMD_NULL'
  10 = 'XTS_CMD_INIT'
  30 = 'XTS_IDLE'
   = ''
END_TEXTLIST

// ---- XTS/_Visualization/XTS_TRANSPORT.TcVIS
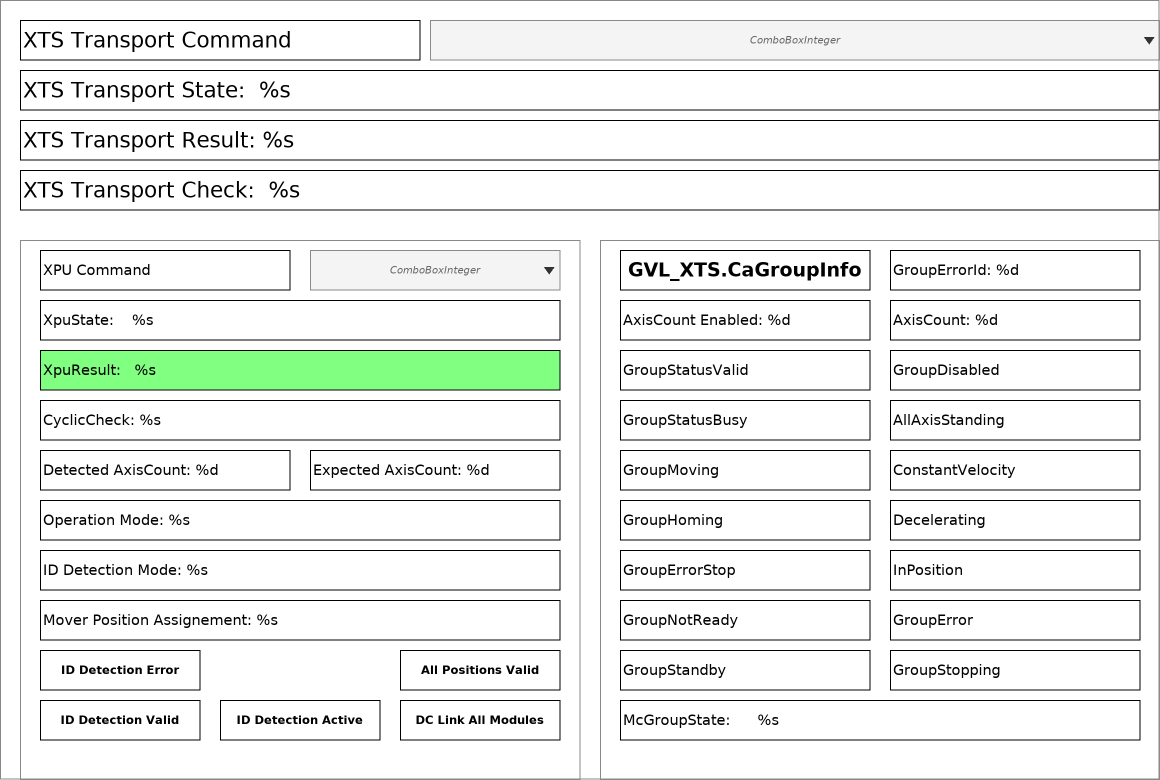
VISUALIZATION XTS_TRANSPORT  // 1160x780
    Rectangle (20,20 400x40), "XTS Transport Command"
    ComboBoxInteger (430,20 730x40), variable: GVL_XTS.XtsTransportCtrl.Cmd, text list: 'TL_E_CTRL_TRANSPORT'
    Frame (20,240 560x540)
        shows XPU_VISU()
    Frame (600,240 560x540)
        shows GROUP_VISU()
    Rectangle (20,70 1140x40), "XTS Transport State: %s", text variable: MAIN.sTransportState
    Rectangle (20,120 1140x40), "XTS Transport Result: %s", text variable: MAIN.sTransportResult
    Rectangle (20,170 1140x40), "XTS Transport Check: %s", text variable: MAIN.sTransportCheck
END_VISUALIZATION

// ---- XTS/_Visualization/XPU_VISU.TcVIS
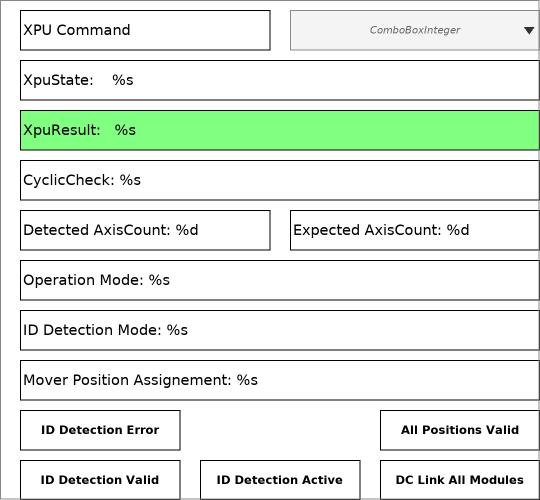
VISUALIZATION XPU_VISU  // 540x500
    Rectangle (20,10 250x40), "XPU Command"
    ComboBoxInteger (290,10 250x40), variable: GVL_XTS.XpuCtrl.Cmd, text list: 'TL_E_CTRL_XPU'
    Rectangle (20,160 520x40), "CyclicCheck: %s", text variable: MAIN.sXpuCheck
    Rectangle (20,60 520x40), "XpuState: %s", text variable: MAIN.sXpuState
    Rectangle (20,110 520x40), "XpuResult: %s", text variable: MAIN.sXpuResult, colour toggle: (MAIN.eXpuResult = E_PROGRESS.PROGRESS_ERROR)
    Rectangle (380,410 160x40), "All Positions Valid", colour toggle: GVL_XTS.XtsTransportState.XpuInfo.AllPositionsValid
    Rectangle (20,410 160x40), "ID Detection Error", colour toggle: GVL_XTS.XtsTransportState.XpuInfo.IdDetectionError
    Rectangle (20,460 160x40), "ID Detection Valid", colour toggle: GVL_XTS.XtsTransportState.XpuInfo.IdDetectionValid
    Rectangle (200,460 160x40), "ID Detection Active", colour toggle: GVL_XTS.XtsTransportState.XpuInfo.IdDetectionActive
    Rectangle (20,260 520x40), "Operation Mode: %s", text variable: MAIN.sXpuOpMode
    Rectangle (20,310 520x40), "ID Detection Mode: %s", text variable: MAIN.sXpuMoverdetectionMode
    Rectangle (20,360 520x40), "Mover Position Assignement: %s", text variable: MAIN.sXpuMoverAssignement
    Rectangle (290,210 250x40), "Expected AxisCount: %d", text variable: GVL_XTS.XtsTransportState.XpuInfo.nExpectedAxisCount
    Rectangle (20,210 250x40), "Detected AxisCount: %d", text variable: GVL_XTS.XtsTransportState.XpuInfo.nDetectedAxisCount
    Rectangle (380,460 160x40), "DC Link All Modules", colour toggle: GVL_XTS.XtsTransportState.XpuState.DcLink
END_VISUALIZATION
